(* Functionsblocks *************************************************)
	rTrigExecute											:	R_TRIG;
	SoERead													:	FB_SoERead_ByDriveRef	:= (tTimeOut := DEFAULT_ADS_TIMEOUT);
(*******************************************************************)
END_VAR
VAR CONSTANT
	ST_IDLE													:	INT := 0;
	ST_PEAKCURRENT											:	INT := 10;
	ST_COSPHI												:	INT := 20;
	ST_ERROR												:	INT := 998;
	ST_RESET												:	INT := 999;
	
	ERR_PEAKCURRENT											:	UDINT := 1;
	ERR_COSPHI												:	UDINT := 2;
END_VAR


(* Init drive ref **************************************************)
	IF AdsAddr.port <> SoERead.stDriveRef.nSlaveAddr
	THEN
		SoERead.stDriveRef.sNetId							:= F_CreateAmsNetId(AdsAddr.netId);
		SoERead.stDriveRef.nSlaveAddr						:= AdsAddr.port;
		SoERead.stDriveRef.nDriveNo							:= Channel;
	END_IF
(* calculate  ******************************************************)
	IF NOT busy
		AND MemParamSet = ActParameterSet
		AND Enable
	THEN
		AbsoluteCurrent										:= TO_REAL(_AbsoluteCurrent * (MemPeakCurrent / 1000)) / 1000;
		ApparentPower										:= SQRT(3) * TO_LREAL(AbsoluteCurrent * AbsoluteVoltage)  / 1000;
		ActivePower											:= ApparentPower * TO_LREAL(MemCosPhi) / 100.0;
		ReactivePower										:= SQRT(EXPT(ApparentPower,2) - EXPT(ActivePower,2));
	END_IF
(* Trigger Execute *************************************************)
	rTrigExecute(CLK := MemParamSet <> ActParameterSet AND Enable);
	
(* get params ******************************************************)
	CASE state OF
	ST_IDLE:	
		IF rTrigExecute.Q
		THEN
			State											:= ST_PEAKCURRENT;
		END_IF
	ST_PEAKCURRENT:	// read P-x-0092 configured peak current
		IF NOT SoERead.bBusy
			AND SoERead.bExecute
		THEN
			state											:= SEL(SoERead.bError, ST_COSPHI, 99);
			ErrorID											:= SEL(SoERead.bError, 0, ERR_PEAKCURRENT);
			ErrorText										:= SEL(SoERead.bError, '', 'Fehler beim Lesen vom Kanal Spitzenstrom');
		END_IF
		SoERead(
			stDriveRef	:= ,  //See init for drive ref
			nIdn		:= Get_P_WORD(ActParameterSet) + 092,
			nElement	:= EC_SOE_ELEMENT_VALUE (* 16#40*),
			pDstBuf		:= ADR(MemPeakCurrent),
			cbBufLen	:= SIZEOF(MemPeakCurrent),
			bExecute	:= State = 10,
			tTimeout	:= ,
			bBusy		=> ,
			bError		=> ,
			iAdsErrId	=> ,
			iSercosErrId=> ,
			dwAttribute	=> );
	ST_COSPHI:	// read P-x-0104 cos phi
		IF NOT SoERead.bBusy
			AND SoERead.bExecute
		THEN
			MemParamSet										:= SEL(SoERead.bError, ActParameterSet, MemParamSet);
			state											:= SEL(SoERead.bError, ST_IDLE, ST_ERROR);
			ErrorID											:= SEL(SoERead.bError, 0, ERR_COSPHI);
			ErrorText										:= SEL(SoERead.bError, '', 'Fehler beim Lesen vom cos phi Parameter');
		END_IF
		SoERead(
			stDriveRef	:= ,  //See init for drive ref
			nIdn		:= Get_P_WORD(ActParameterSet) + 104,
			nElement	:= EC_SOE_ELEMENT_VALUE (* 16#40*),
			pDstBuf		:= ADR(MemCosPhi),
			cbBufLen	:= SIZEOF(MemCosPhi),
			bExecute	:= State = 20,
			tTimeout	:= ,
			bBusy		=> ,
			bError		=> ,
			iAdsErrId	=> ,
			iSercosErrId=> ,
			dwAttribute	=> );
	ST_ERROR:			// wait till Error is quit
		IF ConfirmTrig
		THEN
			ErrorText										:= '';
			ErrorID											:= 0;
			state											:= ST_RESET;
		END_IF
	ST_RESET:		
		IF NOT SoERead.bBusy
			AND NOT SoERead.bError
		THEN
			state											:= ST_IDLE;
		END_IF
		SoERead(
			stDriveRef	:= ,  //See init for drive ref
			nIdn		:= Get_P_WORD(ActParameterSet) + 092,
			nElement	:= EC_SOE_ELEMENT_VALUE (* 16#40*),
			pDstBuf		:= ADR(MemPeakCurrent),
			cbBufLen	:= SIZEOF(MemPeakCurrent),
			bExecute	:= FALSE,
			tTimeout	:= ,
			bBusy		=> ,
			bError		=> ,
			iAdsErrId	=> ,
			iSercosErrId=> ,
			dwAttribute	=> );
	END_CASE
	
	Error		:= state = ST_ERROR;
	Busy		:= state <> 0 OR SoERead.bBusy;
(*******************************************************************)

METHOD PRIVATE get_P_WORD : WORD
VAR_INPUT
	SetNumber			:	INT;
END_VAR
(* Get P-Word dependent of parameter set *)
	IF SetNumber = 0 THEN
		Get_p_WORD			:= P_0_IDN;
	ELSIF SetNumber = 1 THEN
		Get_P_WORD			:= P_1_IDN;
	ELSIF SetNumber = 2 THEN
		Get_P_WORD			:= P_2_IDN;
	ELSIF SetNumber = 3 THEN
		Get_P_WORD			:= P_3_IDN;
	ELSIF SetNumber = 4 THEN
		Get_P_WORD			:= P_4_IDN;
	ELSIF SetNumber = 5 THEN
		Get_P_WORD			:= P_5_IDN;
	ELSIF SetNumber = 6 THEN
		Get_P_WORD			:= P_6_IDN;
	ELSIF SetNumber = 7 THEN
		Get_P_WORD			:= P_7_IDN;
	END_IF
END_METHOD

METHOD PRIVATE get_S_WORD : WORD
VAR_INPUT
	SetNumber			:	INT;
END_VAR
(* Get S-Word dependent of parameter set *)
	IF SetNumber = 0 THEN
		Get_S_WORD			:= S_0_IDN;
	ELSIF SetNumber = 1 THEN
		Get_S_WORD			:= S_1_IDN;
	ELSIF SetNumber = 2 THEN
		Get_S_WORD			:= S_2_IDN;
	ELSIF SetNumber = 3 THEN
		Get_S_WORD			:= S_3_IDN;
	ELSIF SetNumber = 4 THEN
		Get_S_WORD			:= S_4_IDN;
	ELSIF SetNumber = 5 THEN
		Get_S_WORD			:= S_5_IDN;
	ELSIF SetNumber = 6 THEN
		Get_S_WORD			:= S_6_IDN;
	ELSIF SetNumber = 7 THEN
		Get_S_WORD			:= S_7_IDN;
	END_IF
END_METHOD

END_FUNCTION_BLOCK

// POUs/IO/Drives/SoE/AxDriveSoE_Ax5000CommutationCalib
FUNCTION_BLOCK AxDriveSoE_Ax5000CommutationCalib EXTENDS FbBase
VAR CONSTANT
	STEP_COUNT											:	INT := 1;
	P150_NAMEPLATE_TYPE									:	E_AX5000_P_0150_DigitalNamePlate := E_AX5000_P_0150_DigitalNamePlate.EAX5000_P_0150_DIGITALNAMEPLATE_BECKHOFF; //1= Digital nameplate = Beckhoff
	P150_COMMUTATION_MODE_FEEDBACK						:	UINT := 1; //1= Feedback commutation offset
	
//	P150_NO_NAMEPLATE									:	UINT := 0; //0= Digital nameplate = no nameplate
//	P150_COMMUTATION_MODE_ADJUSTABLE					:	UINT := 3; //3= Adjustable mechanical offset 
END_VAR
VAR_OUTPUT CONSTANT
{attribute 'displaymode':='binary'}
	OPTION_READ_ONLY									:	BYTE  := 2#0000_0001; //Read actual commutation offset of the motor (not stored value in drive)
{attribute 'displaymode':='binary'}
	OPTION_P98_IS_EMPTY									:	BYTE  := 2#0000_0010; //Digital nameplate not initialized, skip check if entries. Select this option for first time setup
END_VAR
VAR_INPUT
	AdsAddr												: 	AMSADDR; //Terminal AMS Net Addr.	
	Channel												:	USINT;

{attribute 'displaymode':='binary'}         			
	Options												:	BYTE  := 2#0000_0000; (* Option constants are predefined, so they can accordingly be passed symbolically to the block 
																					.0 = TRUE read only 
																					*)

	
	MaxComPosDifference									:	LREAL := 15.0; //Maximal commutation position offset (Parameter P167, result of command P166)
END_VAR
VAR_IN_OUT
	axis												: AXIS_REF;
END_VAR
VAR_OUTPUT

	P0053												: AX5000_P_0053; // Configured motor type
	P0058												: AX5000_P_0058; // Mechanical commutation offset after command P166
	P0150												: AX5000_P_0150; // Feedback type form startup list
	P0167												: AX5000_P_0167; //Motor and feedback connection check parameter
	P0098												: AX5000_P_0098_beckhoff := (	
															Id_prat_1:= 1113940843,
															Id_prat_2:= 1752131174,	
														//	Name_plate_type := , 
															Version_no:=2,
															Motor_vendor:= 0, //None
															Serial_number:= 999999); //Digital nameplate
	Offset												:	LREAL; //Scaled value

	SercosErrId											: UDINT;
END_VAR
VAR
(*  Memory *****************************************************)
	lastState											: INT := 0;

(*  Timer ******************************************************)
(*  Trigger ****************************************************)

(*  Blocks *****************************************************)
	SoECommand 											: FB_SoEExecuteCommand 	:= (Timeout := t#30s);
	SoEWritePassword 									: FB_SoEWritePassword 	:= (Password :=(strData := 'AX5000', iActualSize := 128, iMaxSize := 128), Timeout := DEFAULT_ADS_TIMEOUT);
	SoEReset											: FB_SoEReset 			:= (Timeout := DEFAULT_ADS_TIMEOUT);
	SoEWrite											: FB_SoEWrite 			:= (Timeout := T#30S);
	SoERead												: FB_SoERead 			:= (Timeout := DEFAULT_ADS_TIMEOUT);
	
(*  Error ******************************************************)
(*  Dummys *****************************************************)
	{attribute 'hide' := ''}
	i,j													: INT := 0;

END_VAR

	(*********************************************************)
	
(* state machine ********************************************************)
	rtExecute(CLK := Execute);
	CASE state OF
	0 : 
		Busy 											:= FALSE;
		
		IF NOT Execute THEN
			Done 										:= FALSE;
			Error 										:= FALSE;
			ErrorID 									:= 0;
			SercosErrId									:= 0;
		END_IF
		IF rtExecute.Q THEN
			IF axis.status.ControlLoopClosed AND NOT Options.1 THEN
				Error 									:= TRUE;
				ErrorID 								:= 19266; //xis is enabled but should not be enabled for this process.

			ELSIF AdsAddr.netId[0] = 0
			THEN
 				Error 									:= TRUE;
				ErrorID 								:= 15; //Invalid AMS net id
	
			ELSIF AdsAddr.port = 0
			THEN
				Error 									:= TRUE;
				ErrorID 								:= 24; //Invalid ADS Port
						
			ELSE
				Busy									:= TRUE;	
				Done 									:= FALSE;
				Error 									:= FALSE;
				ErrorID 								:= 0;
				SercosErrId								:= 0;	
				
				Offset									:= 0.0;
				MEMSET(ADR(P0053),0,SIZEOF(P0053));
				MEMSET(ADR(P0058),0,SIZEOF(P0058));
				MEMSET(ADR(P0150),0,SIZEOF(P0150));
				MEMSET(ADR(P0167),0,SIZEOF(P0167));
				
				SoECommand(Execute := FALSE, Axis := axis);
				SoEWrite(Execute := FALSE, Axis := axis);
				SoERead(Execute := FALSE, Axis := axis);
				SoEReset(Execute := FALSE, Axis := axis);
				SoEWritePassword(Execute := FALSE, Axis := axis);
		
					
				state									:= state + STEP_COUNT;
			END_IF
		END_IF
	
	1:	(*write drive password *)
		SoEWritePassword(
			NetId:= , 
			Execute:=TRUE , 
			Timeout:= , 
			Password:= , //See declaration 
			Axis:=axis , 
			Busy=> , 
			Error=> , 
			AdsErrId=> , 
			SercosErrId=> );
	
		IF NOT SoEWritePassword.busy
		THEN
			IF SoEWritePassword.Error
			THEN
				Busy									:= FALSE;
				Error									:= TRUE;
				ErrorId									:= SoEWritePassword.AdsErrId;
				SercosErrId								:= SoEWritePassword.SercosErrId;
				state 									:= 0;
			ELSE
				
				state									:= state + STEP_COUNT;
			END_IF		
			SoEWritePassword(Execute := FALSE, Axis := axis);
		END_IF
			
	2:	(* Reset active errors *)
		SoEReset(
			NetId:= , 
			Execute:=TRUE , 
			Timeout:= , 
			Axis:=axis , 
			Busy=> , 
			Error=> , 
			AdsErrId=> , 
			SercosErrId=> );
			
		IF NOT SoEReset.Busy
		THEN
			IF SoEReset.Error
			THEN
				Busy									:= FALSE;
				Error									:= TRUE;
				ErrorId									:= SoEReset.AdsErrId;
				SercosErrId								:= SOEReset.SercosErrId;
				state 									:= 0;
			ELSE
				
				state									:= state + STEP_COUNT;
			END_IF	
			SoEReset(Execute := FALSE, Axis := axis);	
		END_IF

	3: // read configured motor type
		SoERead(
			NetId:= , 
			Idn:=P_0_IDN+53 , // IDN P-0-0053 Configured motor type
			Element:=EC_SOE_ELEMENT_VALUE , 
			pDstBuf:=ADR(P0053) , 
			BufLen:=SIZEOF(P0053) , 
			Execute:=TRUE , 
			Timeout:= , 
			Axis:=axis , 
			Busy=> , 
			Error=> , 
			AdsErrId=> , 
			SercosErrId=> , 
			Attribute=> );
			
		IF NOT SoERead.Busy
		THEN
			IF SoERead.Error
			THEN
				Busy									:= FALSE;
				Error									:= TRUE;
				ErrorId									:= SoERead.AdsErrId;
				SercosErrId								:= SoERead.SercosErrId;
				state 									:= 0;
			ELSE		
				
				state									:= state + STEP_COUNT;
			END_IF	
			SoERead(Execute := FALSE, Axis := axis);	
		END_IF
		
	4: //Read feedback type form startup list
		SoERead(
			NetId:= , 
			Idn:=P_0_IDN+150 , 
			Element:=EC_SOE_ELEMENT_VALUE , 
			pDstBuf:=ADR(P0150) , 
			BufLen:=SIZEOF(P0150) , 
			Execute:=TRUE , 
			Timeout:= , 
			Axis:=axis , 
			Busy=> , 
			Error=> , 
			AdsErrId=> , 
			SercosErrId=> , 
			Attribute=> );
			
		IF NOT SoERead.Busy
		THEN
			IF SoERead.Error
			THEN
				Busy									:= FALSE;
				Error									:= TRUE;
				ErrorId									:= SoERead.AdsErrId;
				SercosErrId								:= SoERead.SercosErrId;
				state 									:= 0;
			ELSE				
				state									:= state + STEP_COUNT;
			END_IF		
			SoERead(Execute := FALSE, Axis := axis);
		END_IF		
		
	5: (* Reserved *****************************************************)
		state											:= state + STEP_COUNT;
		
	6: //Read nameplate to check content (must be initialized) *************************
		SoERead(
			NetId:= , 
			Idn:=P_0_IDN+98 , 
			Element:=EC_SOE_ELEMENT_VALUE , 
			pDstBuf:=ADR(P0098) , 
			BufLen:=SIZEOF(P0098) , 
			Execute:=TRUE, 
			Timeout:= , 
			Axis:=axis , 
			Busy=> , 
			Error=> , 
			AdsErrId=> , 
			SercosErrId=> , 
			Attribute=> );	
		
		IF NOT SoERead.Busy
		THEN
			IF SoERead.Error
			THEN
				Busy									:= FALSE;
				Error									:= TRUE;
				ErrorId									:= SoERead.AdsErrId;
				SercosErrId								:= SoERead.SercosErrId;
				state 									:= 0;
			ELSE
				Offset									:= TO_LREAL(P0098.Position_offset) * 0.01;
				SoERead(Execute := FALSE, Axis := axis);	
				//Check parameter of P150
				IF Options.0
				THEN //Read only
					Busy								:= FALSE;
					Done								:= TRUE;
					state 								:= 0;
					
				ELSIF Options.1
				THEN //Nameplate not active, ignore current setting
					state								:= 10;	
					
				ELSIF TO_UINT(P0150.ParameterChannel.CommutationMode0) <> P150_COMMUTATION_MODE_FEEDBACK 
				THEN
					Busy								:= FALSE;
					Error								:= TRUE;
					ErrorId								:= E_AdsErr.DEVICE_INVALIDPARM;
					SercosErrId							:= 16#F749; //Feedback parameter invalid
					state 								:= 0;	
				ELSIF P0150.ParameterChannel.DigitalNamePlate <> P150_NAMEPLATE_TYPE
				THEN
					Busy								:= FALSE;
					Error								:= TRUE;
					ErrorId								:= E_AdsErr.DEVICE_INVALIDPARM;
					SercosErrId							:= 16#F749; //Invalid nameplate
					state 								:= 0;			
			
				ELSIF P0098.Name_plate_type <> P0150.ParameterChannel.DigitalNamePlate 
				THEN
					Busy								:= FALSE;
					Error								:= TRUE;
					ErrorId								:= E_AdsErr.DEVICE_INVALIDPARM;
					SercosErrId							:= 16#F803; //Unknow nameplate
					state 								:= 0;					
				
				ELSIF P0098.Position_offset = 0.0 
				THEN
					Busy								:= FALSE;
					Error								:= TRUE;
					ErrorId								:= E_AdsErr.DEVICE_INVALIDPARM;
					SercosErrId							:= 16#F742; //Invalid commutation offset
					state 								:= 0;
						
				ELSIF P0098.Feedback_typ <> P0150.FeedbackTypeString 
				THEN
					Busy								:= FALSE;
					Error								:= TRUE;
					ErrorId								:= E_AdsErr.DEVICE_INVALIDPARM;
					SercosErrId							:= 16#F708; //Feedback type invalid
					state 								:= 0;		
				ELSIF P0098.Motor_type <> P0053.Configures_motor_type 
				THEN
					Busy								:= FALSE;
					Error								:= TRUE;
					ErrorId								:= E_AdsErr.DEVICE_INVALIDPARM;
					SercosErrId							:= 16#FD09; //Motor type invalid
					state 								:= 0;				
				ELSE
					state								:= 10;	
				END_IF	
			END_IF
		END_IF
		
	10:	// Start command P-0-0160 - calibrate commutation offset ***********************************************	
		SoECommand(
			NetId:='' , 
			Idn:=P_0_IDN+160 , //command P-0-0160 = calibrate commutation offset 
			Execute:= TRUE, 
			Timeout:= , 
			Axis:=axis , 
			Busy=> , 
			Error=> , 
			AdsErrId=> , 
			SercosErrId=> );
		
		IF NOT SoECommand.Busy
		THEN
			IF SoECommand.Error
			THEN
				Busy									:= FALSE;
				Error									:= TRUE;
				ErrorId									:= SoECommand.AdsErrId;
				SercosErrId								:= SoECommand.SercosErrId;
				state 									:= 0;
			ELSE
				state									:= state + STEP_COUNT;
			END_IF		
			SoECommand(Execute := FALSE, Axis := axis);
		END_IF
	
	11: // read mechanical commutation offset result of command P160
		SoERead(
			NetId:= , 
			Idn:=P_0_IDN+58 , // IDN P-0-0167 = parameters to check commutation and rotation direction
			Element:=EC_SOE_ELEMENT_VALUE , 
			pDstBuf:=ADR(P0058) , 
			BufLen:=SIZEOF(P0058) , 
			Execute:= TRUE , 
			Timeout:= , 
			Axis:=axis , 
			Busy=> , 
			Error=> , 
			AdsErrId=> , 
			SercosErrId=> , 
			Attribute=> );	
		
		IF NOT SoERead.Busy
		THEN
			IF SoERead.Error
			THEN
				Busy									:= FALSE;
				Error									:= TRUE;
				ErrorId									:= SoERead.AdsErrId;
				SercosErrId								:= SoERead.SercosErrId;
				state 									:= 0;
			ELSE
				//Init nameplate information - see also declaration
				P0098.Motor_type						:= P0053.Configures_motor_type;
				P0098.Feedback_typ						:= P0150.FeedbackTypeString;	
				P0098.Name_plate_type					:= P0150.ParameterChannel.DigitalNamePlate;
				P0098.Position_offset					:= P0058.Mechanical_commutation_offset;
				Offset									:= TO_LREAL(P0058.Mechanical_commutation_offset) * 0.01;		
	
				state									:= state + STEP_COUNT;
			END_IF	
			SoERead(Execute := FALSE, Axis := axis);	
		END_IF
		
	12: // Start command P-0-0166 - Motor and feedback connection check 
		SoECommand(
			NetId:='' , 
			Idn:=P_0_IDN+166 , //command P-0-0166 = motor and feedback connection check 
			Execute:= TRUE, 
			Timeout:= , 
			Axis:=axis , 
			Busy=> , 
			Error=> , 
			AdsErrId=> , 
			SercosErrId=> );
		
		IF NOT SoECommand.Busy
		THEN
			IF SoECommand.Error
			THEN
				Busy									:= FALSE;
				Error									:= TRUE;
				ErrorId									:= SoECommand.AdsErrId;
				SercosErrId								:= SoECommand.SercosErrId;
				state 									:= 0;
			ELSE
				
				state									:= state + STEP_COUNT;
			END_IF		
			SoECommand(Execute := FALSE, Axis := axis);
		END_IF
	
	13: // read P-0-0167 read connection check results
		SoERead(
			NetId:= , 
			Idn:=P_0_IDN+167 , // IDN P-0-0167 = parameters to check commutation and rotation direction
			Element:=EC_SOE_ELEMENT_VALUE , 
			pDstBuf:=ADR(P0167) , 
			BufLen:=SIZEOF(P0167) , 
			Execute:= TRUE , 
			Timeout:= , 
			Axis:=axis , 
			Busy=> , 
			Error=> , 
			AdsErrId=> , 
			SercosErrId=> , 
			Attribute=> );
				
		IF NOT SoERead.Busy
		THEN
			IF SoERead.Error
			THEN
				Busy									:= FALSE;
				Error									:= TRUE;
				ErrorId									:= SoERead.AdsErrId;
				SercosErrId								:= SoERead.SercosErrId;
				state 									:= 0;
			ELSE				
				IF P0167.EqualDirektions <> 1
					OR
					TO_LREAL(P0167.Commutation_position_difference) * 0.01 > MaxComPosDifference 
					AND TO_LREAL(P0167.Commutation_position_difference) * 0.01 < 360.0 - MaxComPosDifference
				THEN
					Busy								:= FALSE;
					Error								:= TRUE;
					ErrorId								:= E_AdsErr.DEVICE_INVALIDPARM;
					SercosErrId							:= 16#F702; //Feedback position invalid
					state 								:= 0;
				ELSE                                	
					state								:= state + STEP_COUNT;
				END_IF
			END_IF		
			SoERead(Execute := FALSE, Axis := axis);
		END_IF
		
	14:	// Write digital motor plate with commutation offset
		SoEWrite(
			NetId:= , 
			Idn:=P_0_IDN+98, // P0-0-0098 = digital motor plate 
			Element:=EC_SOE_ELEMENT_VALUE , 
			pSrcBuf:=ADR(P0098) ,
			BufLen:=SIZEOF(P0098) ,
			Execute:=TRUE,
			Timeout:= , 
			Password:= SoEWritePassword.Password, 
			Axis:=axis , 
			Busy=> , 
			Error=> , 
			AdsErrId=> , 
			SercosErrId=> );
			
		IF NOT SoEWrite.Busy
		THEN
			IF SoEWrite.Error
			THEN
				Busy									:= FALSE;
				Error									:= TRUE;
				ErrorId									:= SoEWrite.AdsErrId;
				SercosErrId								:= SoEWrite.SercosErrId;
				state 									:= 0;
			ELSE
				
				state									:= state + STEP_COUNT;
			END_IF	
			SoEWrite(Execute := FALSE, Axis := axis);	
		END_IF

	15: // Command P-0-0162 - Save digital name plate
		SoECommand(
			NetId:= , 
			Idn:=P_0_IDN+162 , //save digital name plate 
			Execute:=TRUE , 
			Timeout:= , 
			Axis:=axis , 
			Busy=> , 
			Error=> , 
			AdsErrId=> , 
			SercosErrId=> );
	
		IF NOT SoECommand.Busy
		THEN
			IF SoECommand.Error
			THEN
				Busy									:= FALSE;
				Error									:= TRUE;
				ErrorId									:= SoECommand.AdsErrId;
				SercosErrId								:= SoECommand.SercosErrId;
				state 									:= 0;
			ELSE
				
				state									:= state + STEP_COUNT;
			END_IF		
			SoECommand(Execute := FALSE, Axis := axis);
		END_IF

	16: // Write digital motor plate with commutation offset again
		SoEWrite(
			NetId:= , 
			Idn:=P_0_IDN+98 , 
			Element:=EC_SOE_ELEMENT_VALUE , 
			pSrcBuf:=ADR(P0098) ,
			BufLen:=SIZEOF(P0098) ,
			Execute:= TRUE,
			Timeout:= , 
			Password:=SoEWritePassword.Password  , 
			Axis:=axis , 
			Busy=> , 
			Error=> , 
			AdsErrId=> , 
			SercosErrId=> );
				
		IF NOT SoEWrite.Busy
		THEN
			IF SoEWrite.Error
			THEN
				Busy									:= FALSE;
				Error									:= TRUE;
				ErrorId									:= SoEWrite.AdsErrId;
				SercosErrId								:= SoEWrite.SercosErrId;
				state 									:= 0;
			ELSE
				
				state									:= state + STEP_COUNT;
			END_IF	
			SoEWrite(Execute := FALSE, Axis := axis);	
		END_IF

	17: //Start command P-0-0161 - Save commutation offset in feedback 1
		SoECommand(
			NetId:= , 
			Idn:=P_0_IDN+161 , //save commutation offset 
			Execute:=TRUE , 
			Timeout:= , 
			Axis:=axis , 
			Busy=> , 
			Error=> , 
			AdsErrId=> , 
			SercosErrId=> );
		
		IF NOT SoECommand.Busy
		THEN
			IF SoEWrite.Error
			THEN
				Busy									:= FALSE;
				Error									:= TRUE;
				ErrorId									:= SoEWrite.AdsErrId;
				SercosErrId								:= SoEWrite.SercosErrId;
				state 									:= 0;
			ELSE
				Busy									:= FALSE;
				Done									:= TRUE;
				state 									:= 0;					
			END_IF		
			SoECommand(Execute := FALSE, Axis := axis);
		END_IF
	
	ELSE
		;
	END_CASE

(* Record last state ******************************************)
IF state <> lastState AND state <> 0 AND NOT Error
THEN 
	lastState											:= state;
END_IF

(*************************************************************)

{attribute 'monitoring' := 'call'}
PROPERTY PUBLIC optP98IsEmpty : BOOL
GET
optP98IsEmpty := Options.1;
END_GET
SET
Options.1 := optP98IsEmpty;
END_SET
END_PROPERTY

{attribute 'monitoring' := 'call'}
PROPERTY PUBLIC optReadOnly : BOOL
GET
optReadOnly := Options.0;
END_GET
SET
Options.0 := optReadOnly;
END_SET
END_PROPERTY

END_FUNCTION_BLOCK

// POUs/IO/Drives/SoE/AxDriveSoE_Ax5000Param
{attribute 'no_check'}
//FB template to read and write parameter
//The FB can be enherided and derivatived methods of SeqRead/SeqWrite used for application specific parameter.
//The extended methods need to call the super class at the beginning and return true if execution will be finished. The allowed states for new parameter are 1..99
FUNCTION_BLOCK AxDriveSoE_Ax5000Param EXTENDS AxRWParaBase
VAR_OUTPUT CONSTANT
END_VAR 
VAR_INPUT                               					
	AdsAddr													: 	AMSADDR; //Terminal AMS Net Addr. 
	Channel													:	USINT := 0; //Drive channel 0 or 1 for a two channel AX5000
	SetKvPosition											:	LREAL; //S-0-0104 (rad/s)rad - e.g. 10.0		
	SetKpVelocity											:	LREAL; //S-0-0100 mA/(rad/s) - e.g. 0.058	
	SetTnVelocity											:	LREAL; //S-0-0101 0.1ms 		- e.g. 0.015	
END_VAR 
VAR_IN_OUT
END_VAR                               					
VAR_OUTPUT 	
//	MotorSN													:	STRING(15); 
	KvPosition												:	LREAL;//S-0-0104
	KpVelocity												:	LREAL;//S-0-0100
	TnVelocity												:	LREAL;//S-0-0101
	NominalMainVoltage										:	LREAL;//P-0-0201 Volt 
	ConfiguredChnPeakForce									:	LREAL;//P-0-0094 Nm                    										
	ErrorSoEId												:	UDINT := 0;
END_VAR                         	
VAR
(* Cache ************************************************************)

	
(* Trigger **********************************************************)

(* Timer ******************************************************************)

(* FBs ***************************************************************)
	SoEWrite												: 	FB_SoEWrite_ByDriveRef := (tTimeout := DEFAULT_ADS_TIMEOUT); //SoE read
	SoERead													: 	FB_SoERead_ByDriveRef := (tTimeout := DEFAULT_ADS_TIMEOUT); //SoE wriet

(* Dummy memory **********************************************************)

END_VAR

	(* Read/Write drive parameter														*)
	(************************************************************************************)
	
(* Execute ***************************************************************************************)
	SUPER^();
	
(*************************************************************************************************)

PROPERTY PROTECTED deviceAddrIsValid : BOOL
GET
deviceAddrIsValid := AdsAddr.port > 0;
END_GET
END_PROPERTY

METHOD PROTECTED getValue : BOOL //Return value = TRUE if execution finished and state incremented 
VAR_INPUT
	Idn							:	WORD;
	Element						:	BYTE;
	Len							:	UDINT;
	pActValue					:	PVOID; //Address of variable for actual value
	pSetValue					:	PVOID; //Address of variable for ser value variable, can be zero if no corresponding SetVariable exists
END_VAR

SoERead(bExecute := TRUE, nIdn := Idn, nElement := Element, pDstBuf := pActValue, cbBufLen := Len);
IF NOT SoERead.bBUSY 	
THEN
	IF NOT SoERead.bError
	THEN
		IF pSetValue <> 0 THEN MEMCPY(pSetValue, pActValue, Len); END_IF
		state 												:= state + 1; 
	ELSE
		Busy												:= FALSE;
		Error												:= TRUE;
		ErrorId												:= SoERead.iAdsErrId;
		ErrorSoEId											:= SoERead.iSercosErrId;
		ErrorText											:= CONCAT('Error read parameter in state:' , TO_STRING(state * -1));
		ErrorText											:= CONCAT(ErrorText , CONCAT(' Id:',TO_STRING(ErrorId)));
		ErrorText											:= CONCAT(ErrorText , CONCAT(' Sercos Err :',TO_STRING(ErrorSoEId)));
		State												:= 9999;
	END_IF
	SoERead(bExecute := FALSE);
	getValue												:= TRUE;
END_IF
END_METHOD

METHOD PROTECTED seqRead : BOOL //Return value = TRUE if execution finished 
VAR_IN_OUT
	State							:	INT;
END_VAR

(* Sequence read parameter **********************************)
	CASE state OF
	1..99: //Read application specific parameter  
		SeqRead												:= TRUE;
		
	1001: (* Init step ******************************************************)		
		SoERead(bExecute:=FALSE);
		IF NOT SoERead.bBusy
		THEN
			SoERead.stDriveRef.sNetId						:= F_CreateAmsNetId(AdsAddr.netId);	
			SoERead.stDriveRef.nSlaveAddr 					:= AdsAddr.port;
			SoERead.stDriveRef.nDriveNo 					:= TO_BYTE(Channel);			
			state											:= state + 1;	
		END_IF
		
	1002: (* Kv Position *************************************************************************************)
		IF getValue(Idn:= S_0_IDN + 104,	Element := EC_SOE_ELEMENT_VALUE,	LEN := SIZEOF(_UINT),		pActValue := ADR(_UINT),	pSetValue := 0 )
		THEN
			KvPosition	:= SetKvPosition					:= SEL(Error, TO_LREAL(_UINT) * 0.01, 0.0); 
		END_IF

	1003: (* Kp velocity *******************************************)
		IF getValue(Idn:= S_0_IDN + 100,	Element := EC_SOE_ELEMENT_VALUE,	LEN := SIZEOF(_UDINT),		pActValue := ADR(_UDINT),	pSetValue := 0 )
		THEN
			KpVelocity := SetKpVelocity						:= SEL(Error, TO_LREAL(_UDINT) * 0.001, 0.0);
		END_IF

	1004: (* Tn velocity ********************************************)
		IF getValue(Idn:= S_0_IDN + 101,	Element := EC_SOE_ELEMENT_VALUE,	LEN := SIZEOF(_UINT),		pActValue := ADR(_UINT),	pSetValue := 0 )
		THEN
			TnVelocity	:= SetTnVelocity					:= SEL(Error, TO_LREAL(_UINT) * 0.1, 0.0);
		END_IF
					
	1005: (* Nominal main voltage  ********************************************)
  		IF getValue(Idn:= P_0_IDN + 201,	Element := EC_SOE_ELEMENT_VALUE,	LEN := SIZEOF(_UINT),		pActValue := ADR(_UINT),	pSetValue := 0 )
		THEN
			NominalMainVoltage								:= SEL(Error, TO_LREAL(_UINT) * 0.1, 0.0);
		END_IF	
		
	1006: (* Configured Channel Peak Current ********************************************)
  		IF getValue(Idn:= P_0_IDN + 94,		Element := EC_SOE_ELEMENT_VALUE,	LEN := SIZEOF(_UDINT),		pActValue := ADR(_UDINT),	pSetValue := 0 )
		THEN
			ConfiguredChnPeakForce 							:= SEL(Error, TO_LREAL(_UDINT) * 0.01, 0.0);
		END_IF
	ELSE
		state												:= 1;
	END_CASE

(***********************************************************************************)
END_METHOD

METHOD PROTECTED seqWrite : BOOL //Return value = TRUE if execution finished 
VAR_IN_OUT
	State							:	INT;
END_VAR
(* Sequence write parameter *********************************************)
	CASE state OF
	1..99: //Write application specific parameter  
		SeqWrite											:= TRUE;
		
	1001: (* Init step ******************************************************)		
		SoEWrite(bExecute:= TRUE);
		IF NOT SoEWrite.bBusy
		THEN
			SoEWrite.stDriveRef.sNetId						:= F_CreateAmsNetId(AdsAddr.netId);	
			SoEWrite.stDriveRef.nSlaveAddr 					:= AdsAddr.port;
			SoEWrite.stDriveRef.nDriveNo 					:= Channel;		
			state											:= state + 1;	
		END_IF
	
	1002: (* Kv position *************************************************************************************)
		_UINT												:= TO_UINT(SetKvPosition * 100.0);
		IF setValue(Idn := S_0_IDN + 104, Element := EC_SOE_ELEMENT_VALUE,	LEN := SIZEOF(_UINT),		pActValue := 0,		pSetValue := ADR(_UINT) )
		THEN
			KvPosition										:= SetKvPosition;
		END_IF		
		
	1003: (* Kp velocity ****************************************)
		_UDINT												:= TO_UDINT(SetKpVelocity * 1000.0);
		IF setValue(Idn := S_0_IDN + 100, Element := EC_SOE_ELEMENT_VALUE,	LEN := SIZEOF(_UDINT),		pActValue := 0,		pSetValue := ADR(_UDINT) )
		THEN
			KpVelocity										:= SetKpVelocity;
		END_IF	
		
	1004: (* Tn velocity **********************************)
		_UINT											:= TO_UINT(SetTnVelocity * 10.0);
		IF setValue(Idn := S_0_IDN + 101, Element := EC_SOE_ELEMENT_VALUE,	LEN := SIZEOF(_UINT),		pActValue := 0,		pSetValue := ADR(_UINT) )
		THEN
			TnVelocity										:= SetTnVelocity;
		END_IF		ELSE
		state												:= 1;
	END_CASE

(************************************************************************************)
END_METHOD

METHOD PROTECTED setValue : BOOL //Return value = TRUE if execution finished and state incremented 
VAR_INPUT
	Idn							:	WORD;
	Element						:	BYTE;
	Len							:	UDINT;
	pActValue					:	PVOID; //Address of variable for actual value, can be zero if no corresponding acual value variable exists
	pSetValue					:	PVOID; //Address of variable for set value variable
END_VAR

IF pActValue <> 0 AND pSetValue <> 0 AND_THEN MEMCMP(pSetValue, pActValue, Len) = 0
THEN //Skip write parameter if set and actual value are equel
	state													:= state + 1;	
	setValue												:= TRUE;
ELSE
	SoEWrite(bExecute:= TRUE, nIdn := Idn, nElement := Element, pSrcBuf := pSetValue, cbBufLen := LEN);
	IF NOT SoEWrite.bBusy
	THEN
		IF NOT SoEWrite.bError
		THEN
			IF pActValue <> 0 THEN MEMCPY(pActValue, pSetValue, Len); END_IF	
			state											:= state + 1;
		ELSE
			Busy											:= FALSE;
			Error											:= TRUE;
			ErrorId											:= SoEWrite.iAdsErrId;
			ErrorSoEId										:= SoEWrite.iSercosErrId;
			ErrorText										:= CONCAT('Error write parameter in state:' , TO_STRING(state * -1));
			ErrorText										:= CONCAT(ErrorText , CONCAT(' Id:',TO_STRING(ErrorId)));
			ErrorText										:= CONCAT(ErrorText , CONCAT(' Sercos Err :',TO_STRING(ErrorSoEId)));
			State											:= 9999;
		END_IF
		SoEWrite(bExecute := FALSE);
		setValue											:= TRUE;
	END_IF		
END_IF
END_METHOD

END_FUNCTION_BLOCK

// POUs/IO/Drives/SoE/AxDriveSoE_Ax5000SwitchParamSet
FUNCTION_BLOCK AxDriveSoE_Ax5000SwitchParamSet EXTENDS FbBase
VAR_INPUT
	rAxis													:	REFERENCE TO AXIS_REF := 0; 	// Axis Ref
	TimeOut													:	TIME := DEFAULT_ADS_TIMEOUT;	// Timeout time
	NewParamSet												:	INT;							// Value for new parameterset
END_VAR
VAR_IN_OUT	
(* important for function *)	
	AdsAddr													:	AMSADDR;						// AdsAddr of AX5000
	Channel													:	USINT;                          // Drive channel number
END_VAR
VAR_OUTPUT
	ErrorText												:	T_MaxString;					// Error Text
	ActParamSet												:	INT := -1; 						// Value of active parameter set
END_VAR
VAR
(* Memory **********************************************************)
	StartSwitchParamSet										:	INT := 0;
	
	CountError												:	USINT;
(* Timer ***********************************************************)
	TimerWait												:	TON;
	TimerTimeOut											:	TON;
	
(* Functionsblocks *************************************************)

	SoEWrite												:	FB_SoEWrite_ByDriveRef	:= (tTimeOut := DEFAULT_ADS_TIMEOUT);
	SoERead													:	FB_SoERead_ByDriveRef	:= (tTimeOut := DEFAULT_ADS_TIMEOUT);
(*******************************************************************)
END_VAR
VAR CONSTANT
	ST_IDLE													:	INT := 0;
	ST_REFRESH												:	INT := 10;
	ST_PRESELECT											:	INT := 100;
	ST_DISABLED												:	INT := 110;
	ST_RESETEXECUTE											:	INT := 120;
	ST_SETPARAM												:	INT := 130;
	ST_WAIT													:	INT := 140;
	ST_ERROR												:	INT := 998;
	ST_RESET												:	INT := 999;
	
	ERR_REFRESH												:	UDINT := 1;
	ERR_PRESELECT											:	UDINT := 2;
	ERR_TIMEOUT_DISABLED									:	UDINT := 3;
	ERR_RESETEXECUTE										:	UDINT := 4;
	ERR_EXECUTE												:	UDINT := 5;
	
	PT_WAIT_TIME											:	TIME := T#20MS;
END_VAR

(* abort function-call if the reference is invalid *****************)
	IF NOT __ISVALIDREF(rAxis) THEN
		Busy												:= NOT Error;
		Error												:= TRUE;
		ErrorId												:= 16#4B30;
		ErrorText											:= 'Referenz rAxis invalid (0)';
		RETURN;
	END_IF

(* Init drive ref **************************************************)
	IF AdsAddr.port <> SoERead.stDriveRef.nSlaveAddr
	THEN
		SoERead.stDriveRef.sNetId							:= F_CreateAmsNetId(AdsAddr.netId);
		SoERead.stDriveRef.nSlaveAddr						:= AdsAddr.port;
		SoERead.stDriveRef.nDriveNo							:= Channel;
		
		SoEWrite.stDriveRef									:= SoERead.stDriveRef;
	END_IF
(* Trigger Execute *************************************************)
	rtExecute(CLK := Execute);
	
(* switch parameter set ********************************************)
	CASE State OF
	ST_IDLE:			// wait for command
	(* Get actual parameter set after restart *)
		IF ActParamSet < 0 
		THEN
			State											:= ST_REFRESH;
	(* Start switch parameter set *)
		ELSIF rtExecute.Q
		THEN
			setNewParam(NewParamSet);
		ELSIF NOT Execute
		THEN
			Error											:= FALSE;
			Done											:= FALSE;
			Busy											:= TRUE;
			ErrorId											:= 0;
			ErrorTExt										:= '';
		END_IF
		
	ST_REFRESH: 		// Refresh ActParamSet Variable
		IF NOT SoERead.bBusy
			AND SoERead.bExecute
		THEN
			State											:= SEL(SoERead.bError, ST_IDLE, ST_ERROR);
			Done											:= State = ST_IDLE;
			Error											:= State = ST_ERROR;	
			ErrorID											:= SEL(SoERead.bError, 0, ERR_REFRESH);
			ErrorText										:= SEL(SoERead.bError, '', 'Fehler beim Aktualisieren des aktuellen Parametersatzes');
		END_IF
		
		SoERead(
			stDriveRef	:= ,  //See init for drive ref
			nIdn		:= S_0_IDN + 254,
			nElement	:= EC_SOE_ELEMENT_VALUE (* 16#40*),
			pDstBuf		:= ADR(ActParamSet),
			cbBufLen	:= SIZEOF(ActParamSet),
			bExecute	:= State = ST_REFRESH,
			tTimeout	:= ,
			bBusy		=> ,
			bError		=> ,
			iAdsErrId	=> ,
			iSercosErrId=> ,
			dwAttribute	=> );
			
		ST_PRESELECT:		// Set New param value in drive preselection
			IF NewParamSet = ActParamSet
			THEN
				State										:= ST_IDLE;
			ELSIF NOT SoEWrite.bBusy
				AND SoEWrite.bExecute
			THEN
				State										:= SEL(SoEWrite.bError, ST_DISABLED, ST_ERROR);
				ErrorID										:= SEL(SoERead.bError, 0, ERR_PRESELECT);
				ErrorText									:= SEL(SoERead.bError, '', 'Fehler beim Schreiben der Vorwahl');
			END_IF
			
			SoEWrite(
				stDriveRef	:= ,  //See init for drive ref
				nIdn		:= S_0_IDN + 217,
				nElement	:= EC_SOE_ELEMENT_VALUE (* 16#40*),
				pSrcBuf		:= ADR(NewParamSet),
				cbBufLen	:= SIZEOF(NewParamSet),
				bExecute	:= State = ST_PRESELECT,
				tTimeout	:= ,
				bBusy		=> ,
				bError		=> ,
				iAdsErrId	=> ,
				iSercosErrId=> );
				
		ST_DISABLED:		// check if axis is disabled
			TimerTimeOut(IN := NOT rAxis.Status.Disabled, PT := TimeOut);
			IF TimerTimeOut.Q THEN
				TimerTimeOut(IN := FALSE);
				State											:= ST_ERROR;
				ErrorID											:= SEL(SoERead.bError, 0, ERR_TIMEOUT_DISABLED);
				ErrorText										:= SEL(SoERead.bError, '', 'Achse ist nicht deaktiviert');
			ELSIF rAxis.Status.Disabled THEN
				TimerTimeOut(IN := FALSE);
				State											:= ST_RESETEXECUTE;
			END_IF
		
		ST_RESETEXECUTE:	// reset the execute command in drive	
			StartSwitchParamSet									:= 0;
			IF NOT SoEWrite.bBusy
				AND SoEWrite.bExecute
			THEN
				State											:= SEL(SoEWrite.bError, ST_SETPARAM, ST_ERROR);
				ErrorID											:= SEL(SoERead.bError, 0, ERR_RESETEXECUTE);
				ErrorText										:= SEL(SoERead.bError, '', 'Fehler beim Zurücksetzen des Ausführungskomamando');
			END_IF
			SoEWrite(
				stDriveRef	:= ,  //See init for drive ref
				nIdn		:= S_0_IDN + 216,
				nElement	:= EC_SOE_ELEMENT_VALUE (* 16#40*),
				pSrcBuf		:= ADR(StartSwitchParamSet),
				cbBufLen	:= SIZEOF(StartSwitchParamSet),
				bExecute	:= State = ST_RESETEXECUTE,
				tTimeout	:= ,
				bBusy		=> ,
				bError		=> ,
				iAdsErrId	=> ,
				iSercosErrId=> );		
				
		ST_SETPARAM:		// Execute switch parameter set
			StartSwitchParamSet								:= 3;
			IF NOT SoEWrite.bBusy
				AND SoEWrite.bExecute
			THEN
				State										:= SEL(SoEWrite.bError, ST_WAIT, ST_ERROR);
				ErrorID										:= SEL(SoERead.bError, 0, ERR_EXECUTE);
				ErrorText									:= SEL(SoERead.bError, '', 'Fehler beim Setzen des Ausführungskommandos');
			END_IF
			SoEWrite(
				stDriveRef	:= ,  //See init for drive ref
				nIdn		:= S_0_IDN + 216,
				nElement	:= EC_SOE_ELEMENT_VALUE (* 16#40*),
				pSrcBuf		:= ADR(StartSwitchParamSet),
				cbBufLen	:= SIZEOF(StartSwitchParamSet),
				bExecute	:= State = ST_SETPARAM,
				tTimeout	:= ,
				bBusy		=> ,
				bError		=> ,
				iAdsErrId	=> ,
				iSercosErrId=> );
				
		ST_WAIT:			// wait a short time while the drive works with the command
			TimerWait(IN := TRUE, pt := PT_WAIT_TIME);
			IF TimerWait.Q THEN
				TimerWait(IN := FALSE);
				State										:= ST_REFRESH;
			END_IF
			
		ST_ERROR:			// wait till Error is quit
			IF TRUE
			THEN
				State										:= ST_RESET;
			END_IF
			
		ST_RESET:			// Reset Error			
			State											:= ST_IDLE;
			SoEWrite(
				stDriveRef	:= ,  //See init for drive ref
				nIdn		:= S_0_IDN + 216,
				nElement	:= EC_SOE_ELEMENT_VALUE (* 16#40*),
				pSrcBuf		:= ADR(StartSwitchParamSet),
				cbBufLen	:= SIZEOF(StartSwitchParamSet),
				bExecute	:= FALSE,
				tTimeout	:= ,
				bBusy		=> ,
				bError		=> ,
				iAdsErrId	=> ,
				iSercosErrId=> );
			SoERead(
				stDriveRef	:= ,  //See init for drive ref
				nIdn		:= S_0_IDN + 254,
				nElement	:= EC_SOE_ELEMENT_VALUE (* 16#40*),
				pDstBuf		:= ADR(ActParamSet),
				cbBufLen	:= SIZEOF(ActParamSet),
				bExecute	:= FALSE,
				tTimeout	:= ,
				bBusy		=> ,
				bError		=> ,
				iAdsErrId	=> ,
				iSercosErrId=> ,
				dwAttribute	=> );
	END_CASE
	Busy													:= State <> ST_IDLE ;
(*******************************************************************)

METHOD setNewParam : BOOL	// Result = Busy
VAR_INPUT
	ParamNo					:	INT;
END_VAR

	IF ParamNo <> ActParamSet
		AND State = ST_IDLE
	THEN
		Error											:= FALSE;
		Done											:= FALSE;
		Busy											:= TRUE;
		ErrorId											:= 0;
		ErrorTExt										:= '';
		NewParamSet 									:= ParamNo;
		TimerWait(IN := FALSE);
		TimerTimeOut(IN := FALSE);
		State											:= ST_PRESELECT;
	END_IF
	
	SetNewParam											:= State <> ST_IDLE;
END_METHOD

END_FUNCTION_BLOCK

// POUs/IO/Drives/SoE/AxDriveSoE_Ax5000wEvents
{attribute 'no_check'}
//AX5000 SoE status and diagnosis FB with eventlogger 
FUNCTION_BLOCK AxDriveSoE_Ax5000wEvents EXTENDS AxDriveSoE_Ax5000
VAR_INPUT
	EnableEvent												:	BOOL := TRUE;
	ConfirmTrig												:	BOOL ;
	SourceId												:	UDINT := 102000; //SoE Drive default multisource Id + Ax id
	Name													:	STRING(30) := '';
	ErrorLimitPos											:	BOOL := FALSE;
	ErrorLimitNeg											:	BOOL := FALSE;
END_VAR                 									
VAR_IN_OUT              									
END_VAR                 									
VAR_OUTPUT              	                    										
	EventStatus												:	DWORD;
	NoOfActiveEvents										:	INT;
	Error													: 	BOOL; //ADS error SoE FBs
{attribute 'displaymode':='hex'}
	ErrorId													:	UDINT; //ADS error id of SoE FBs
	ErrorText												: 	STRING(40);
END_VAR
VAR_OUTPUT CONSTANT
END_VAR
VAR

(* Zwischenspeicher *********************************************************************)


(* Timer ********************************************************************************)

(* Trigger ******************************************************************************)

(* Bausteine ****************************************************************************)
	Event													:	EventHandlingGrp10;

(* Dummy Speicher **********************************************************)
	i														: INT := 0 ;


(****************************************************************************)
END_VAR

	(************************************************************************************)
	(*																					*)
	(*		B E C K H O F F   N E W   A U T O M A T I O N   T E C H N O L O G Y    		*)
	(*																					*)
	(*		Eiserstr.5	D-33415 Verl	Germany	phone:	+49-5246-0	www.Beckhoff.Com	*)
    (*																					*)
    (*		Bausteinbeschreibung	:	AX5000 Drive Ctrl								*)
	(*		TwinCAT-Version			:	3.x or higher 									*)
	(*		Version					:	V3.0 											*)
 	(*		Autor					:	Daniel Schlingmann								*)
	(*		Lib						:	TcMc2Drive.lib / TcDrive.Lib					*)
	(*																					*)
	(************************************************************************************)

(* Trigger reset if by active quit **********)
	IF ConfirmTrig
	THEN
		confirm();
	END_IF

(* Call super *****************************)
	SUPER^();
	
(* Call events ****************************************************)
	_callEvents();

(******************************************************************************)

METHOD PRIVATE _callEvents : BOOL
VAR_INPUT
END_VAR

(* Check if msg activ and init some parameter ***********************)
	IF Event.no[1].Text2 <> Name AND Name <> '' OR Event.no[1].Text2 = '' AND rAxis.NcToPlc.AxisId <> 0
	THEN
		Event.no[1].eClass 									:= TC2_SYSTEM.TCEVENTCLASS_HINT;

		(* Init Name *)
		FOR i := Event.MIN_EVENT TO Event.MAX_EVENT DO
			Event.no[i].Text2								:= SEL(LEN(name)>1,CONCAT('Axis id:',DWORD_TO_STRING(rAxis.NcToPlc.AxisId)),name);
		END_FOR
	END_IF

(* workl Event Ctrl *************************************************)
	Event(
		ConfirmTrig := ConfirmTrig,
		Disable		:= rAxis.NcToPlc.AxisId = 0 OR NOT EnableEvent,
		SourceId	:= SourceId + rAxis.NcToPlc.AxisId,
		Status		=> EventStatus,
		NoOfActiveEvents => NoOfActiveEvents);

(* Error Hdl FB ******************************************************************)
	IF rAxis.Status.OpMode.SimulationAxis OR Event.confirmTrig
	THEN
		;
	ELSIF SoEDriveReset.bError
	THEN
		Error												:=	TRUE;
		ErrorId												:= 0;
		SercosErrorId										:= SoEDriveReset.iSercosErrId;
		ErrorText											:= CONCAT('SoeDrvReset SercosErrId: ',DWORD_TO_HEXSTR(SoEDriveReset.iSercosErrId,4,FALSE));
		ErrorText											:=	CONCAT(CONCAT(ErrorText,', ADSErrId: '),UINT_TO_STRING(SoEDriveReset.iAdsErrId));
	ELSIF SoEAX5000SetMotorCtrlWord.bError
	THEN
		Error												:=	TRUE;
		ErrorId												:= 0;
		SercosErrorId										:= SoEAX5000SetMotorCtrlWord.iSercosErrId;
		ErrorText											:= CONCAT('SoESetMotorCtrlWord SercosErrId: ',DWORD_TO_HEXSTR(SoEAX5000SetMotorCtrlWord.iSercosErrId,4,FALSE));
		ErrorText											:=	CONCAT(CONCAT(ErrorText,', ADSErrId: '),UINT_TO_STRING(SoEAX5000SetMotorCtrlWord.iAdsErrId));
	ELSIF SoERead.bError
	THEN
		Error												:=	TRUE;
		ErrorId												:= 0;
		SercosErrorId										:= SoERead.iSercosErrId;
		ErrorText											:= CONCAT('SoERead SercosErrId: ',DWORD_TO_HEXSTR(SoERead.iSercosErrId ,4,FALSE));
		ErrorText											:=	CONCAT(CONCAT(ErrorText,', ADSErrId: '),UINT_TO_STRING(SoERead.iAdsErrId));
	END_IF

(* Event Logger Meldungen *****************************************************)
	Event.no[1].Flag 										:= Status.bNotReadyToPowerUp;
	Event.no[2].Flag 										:= Status.bDrvShutdownBitC1D AND stateReadStatus = 0; Event.no[2].pText3 := ADR(DiagMsg.strData);
	Event.no[3].Flag 										:= FALSE;
	Event.no[4].Flag 										:= ErrorLimitPos;
	Event.no[5].Flag 										:= ErrorLimitNeg;
	Event.no[6].Flag 										:= SafetyError AND DiagNumber <> 16#0000_FDD9;
	Event.no[7].Flag 										:= FALSE;
	Event.no[8].Flag 										:= FALSE;
	Event.no[9].Flag 										:= FALSE;
	Event.no[10].Flag 										:= Error; Event.no[10].Text1 := TO_STRING(ErrorId);
	
(************************************************************************)
END_METHOD

METHOD PUBLIC confirm : BOOL //Return value = TRUE if busy
VAR_INPUT
END_VAR
Event.confirm();
Error												:= FALSE;
ErrorId												:= 0;
SercosErrorId										:= 0;
ErrorText											:= '';
		
confirm 											:= SUPER^.reset();
END_METHOD

END_FUNCTION_BLOCK

// POUs/IO/Drives/SoE/AxDriveSoE_Rexroth
{attribute 'no_check'}
//Bosch Rexroth EtherCAT SoE Drive Control
//based on Tc2_Drive
FUNCTION_BLOCK AxDriveSoE_Rexroth EXTENDS AxDriveBase
VAR_INPUT
	EnableEvent												:	BOOL := TRUE;
	ResetTrig												:	BOOL := FALSE; (* Quit event and reset drive (SoE Reset) *)
	SourceId												:	UDINT := 102000; //SoE Drive default multisource Id + Ax id
	Name													:	STRING(30) := '';
	ErrorLimitPos											:	BOOL := FALSE;
	ErrorLimitNeg											:	BOOL := FALSE;
	BreakUnlock												:	BOOL := FALSE; //Not implemented yet
	BreakLock												:	BOOL := FALSE; //Not implemented yet					
	SetReferenz												: 	BOOL := FALSE;
	Referenzpos												: 	LREAL := 0.0;
END_VAR                                 					
VAR_IN_OUT                              					
END_VAR                                 					
VAR_OUTPUT                                                					
	InReferenz												:	BOOL; (* Drive in reference *)
	RT_StatusChanged										:	BOOL;                                    						
	Status													:	ST_IndraDriveCsDriveStatus;
	C1D														:	ST_IndraDriveCs_C1D;
	DiagMsg 												: 	ST_SoE_String;
	DiagNumber 												: 	UDINT;
	Operational												: INPUT := (Force := TRUE);	(* Link to ALWAYS_TRUE or operational signal from drive *)
	EcState											AT %I* 	: 	UINT; (* Ethercat InfoData State *)
	SercosErrorId											:	UINT;                    					
	SafetyError										AT %I*	:	BOOL;	(* Ax5805 Drive Safety Error - Bit .7 in Input Safe Data Byte 0 oder 2 *)	
	EventStatus												:	DWORD;
	NoOfActiveEvents										:	INT;
	Busy													:	BOOL;
	Error													:	BOOL;
{attribute 'displaymode':='hex'}
	ErrorId													:	UDINT;
	ErrorText												:	STRING(40);
END_VAR                  						
VAR_OUTPUT CONSTANT
END_VAR
VAR (* EA Internal *)
	EcInfoDataState									AT %I* 	: 	UINT; (* Ethercat InfoData State *)
END_VAR
VAR

(* Cache *********************************************************************)
	MemDriveStatusword										: 	WORD;
	MEM_StatusTrig											:	BYTE;
	StatusTrig												:	BYTE;
	stateReadStatus											:	INT;
	stateCtrl												:	INT := 0;

(* Timer ********************************************************************************)

(* Trigger ******************************************************************************)

(* Instance ****************************************************************************)
	SoEDriveReset											: 	FB_SoEReset := (Timeout		:= DEFAULT_ADS_TIMEOUT);
	SoEWrite												: 	FB_SoEWrite := (Timeout		:= DEFAULT_ADS_TIMEOUT);
	SoERead													: 	FB_SoERead := (Timeout		:= DEFAULT_ADS_TIMEOUT);
	SoEExecuteCmd											:	FB_SoEExecuteCommand := (Timeout		:= DEFAULT_ADS_TIMEOUT);
	EcSetSlaveSTATE											:	FB_EcSetSlaveSTATE := (tTimeout		:= DEFAULT_ADS_TIMEOUT);
	Event													:	EventHandlingGrp10;

(* Dummy Speicher **********************************************************)
	i														: 	INT := 0 ;
	_word													:	WORD;
	_DWORD													:	DWORD;

(****************************************************************************)
END_VAR

	(************************************************************************************)
	(*																					*)
	(*		B E C K H O F F   N E W   A U T O M A T I O N   T E C H N O L O G Y    		*)
	(*																					*)
	(*		Eiserstr.5	D-33415 Verl	Germany	phone:	+49-5246-0	www.Beckhoff.Com	*)
    (*																					*)
    (*		Bausteinbeschreibung	:	Ethercat SoE MC2 Drive Ctrl						*)
	(*		TwinCAT-Version			:	3.x or higher	 								*)
	(*		Version					:	V3.0/05/11										*)
 	(*		Autor					:	Daniel Schlingmann								*)
	(*		Lib						:	TcMC2Drive.lib / TcDrive.Lib					*)
	(*																					*)
	(* Call cyclic																		*)
	(************************************************************************************)

(* abort function-call if the reference is invalid *****************************)
IF NOT __ISVALIDREF(rAxis)  
THEN
	Busy													:= NOT Error;
	Fault													:= TRUE;
	Ready													:= FALSE;
	Error													:= TRUE;
	ErrorId													:= 16#4B30;
	ErrorText												:= 'Referenz rAxis invalid (0)';
	SercosErrorId											:= 0;
	RETURN;
END_IF

(* DriveStatusword *****************************)
	Status 													:= F_ConvWordToSTIndraDriveCsDriveStatus(StatusWord);
	IF rAxis.Status.OpMode.SimulationAxis or AdsAddr.port = 0
	THEN
		Status.bNotReadyToPowerUp							:= FALSE;	
		Status.bDrvShutdownBitC1D							:= FALSE;
		Status.bReadyForEnable								:= TRUE;
		Status.bEnabled										:= TRUE;	
	END_IF
	
(* Drive Operation Input ***********************)
	Operational(
		Force		:= rAxis.Status.OpMode.SimulationAxis ,
		Invert		:= ,
		PT_ON		:= ,
		PT_OFF		:= ,
		Q_DIRECT	=> ,
		Q			=> ,
		Q_RT		=> ,
		Q_FT		=> );

(* DriveStatusBits ***********************************************)
	Fault													:= Status.bDrvShutdownBitC1D
																OR rAxis.NcToPlc.StateDWord.28 (* DriveDeviceError *)
																OR rAxis.NcToPlc.StateDWord.30; (* IODataInvalid *)
                                						
	Ready 													:= NOT Fault
																	AND(Status.bReadyForEnable OR Status.bEnabled)
																	AND Operational.Q;
  
	SwitchedOn												:= Status.bEnabled AND NOT Fault;	
	                              	
(* Reset Drive ****************************************************)
	SoEDriveReset(
		NetId		:= ,
		Execute		:= ,
		Timeout		:= ,
		Axis		:= rAxis,
		Busy		=> ,
		Error		=> ,
		AdsErrId	=> ,
		SercosErrId	=> );

	IF SoEDriveReset.Busy 
	THEN
		; (* Block ist currend working *)
	ELSIF ResetTrig
	THEN
		reset();
	ELSIF SoEDriveReset.Execute
	THEN
	(*	RefreshStatus();  *)
		SoEDriveReset.Execute 								:= FALSE;
	END_IF

(* Set Etehrcat State to OP ********************************************)
	EcSetSlaveSTATE(
		sNetId		:= F_CreateAmsNetId(nIds := AdsAddr.netId),
		nSlaveAddr	:= AdsAddr.port,
		bExecute	:= ,
		tTimeout	:= ,
		reqState	:= Tc2_EtherCAT.EC_DEVICE_STATE_OP,
		bBusy		=> ,
		bError		=> ,
		nErrId		=> ,
		currState	=> );

	IF EcSetSlaveSTATE.bBusy
	THEN
		; (* Block ist currend working *)
	ELSIF EcSetSlaveSTATE.bExecute
		AND NOT ResetTrig
	THEN
		RefreshStatus();
		EcSetSlaveSTATE.bExecute 							:= FALSE;
	END_IF

(* Referenzieren *******************************************************)
	CASE stateCtrl OF
	-1,0:
		IF SetReferenz AND NOT rAxis.Status.OpMode.SimulationAxis AND AdsAddr.port > 0
		THEN
			writeReferenz();
		ELSE
			stateCtrl										:= 0;
		END_IF

	1: (* Referezwert schreiben **************************************)
		IF NOT SoEWrite.Busy
			AND SoEWrite.Execute
		THEN
			IF SoEWrite.Error
			THEN
				stateCtrl 									:= 0;
			ELSE                							
				stateCtrl									:= 2;
			END_IF
		END_IF

		_DWORD 												:= LREAL_TO_UDINT(Referenzpos);

		SoEWrite(
			NetId		:= ,
			Idn			:= S_0_IDN + 52,
			Element		:= EC_SOE_ELEMENT_VALUE ,
			pSrcBuf		:= ADR(_DWORD),
			BufLen		:= SIZEOF(_DWORD),
			Execute		:= stateCtrl = 1,
			Timeout		:= ,
			Password	:= ,
			Axis		:= rAxis,
			Busy		=> ,
			Error		=> ,
			AdsErrId	=> ,
			SercosErrId	=> );

	2: (* commad for setting setvalue *)
		IF NOT SoEExecuteCmd.Busy
			AND SoEExecuteCmd.Execute
		THEN
			IF SoEExecuteCmd.Error
			THEN
				stateCtrl 									:= 0;
			ELSE
				RefreshStatus();
				IF NOT SetReferenz
				THEN
					stateCtrl 								:= 0;
				ELSE            							
					stateCtrl 								:= -1;
				END_IF
			END_IF
		END_IF

		SoEExecuteCmd(
			NetId		:= '',
			Idn			:= P_0_IDN + 12,
			Execute		:= stateCtrl = 2,
			Timeout		:= ,
			Axis		:= rAxis,
			Busy		=> ,
			Error		=> ,
			AdsErrId	=> ,
			SercosErrId	=> );
	ELSE
		;
	END_CASE


(* evaluate sercos DriveStatusword *********************************************************)
	RT_StatusChanged 										:= SHR(StatusWord,2) <> MemDriveStatusword;
	MemDriveStatusword 										:= SHR(StatusWord,2);

(* Start Read Drive status *****************************************************************)
	CASE stateReadStatus OF
	0:
		StatusTrig.0 										:= rAxis.NcToPlc.StateDWord.28; (* DriveDeviceError *)
		StatusTrig.1 										:= rAxis.NcToPlc.StateDWord.30; (* IODataInvalid *)
                                							
		IF NOT rAxis.Status.OpMode.SimulationAxis AND AdsAddr.port > 0
			AND(RT_StatusChanged OR MEM_StatusTrig <> StatusTrig)
		THEN
			RefreshStatus();
		ELSE
			;
		END_IF

	(* Read Class 1 Diag *********************************************************)
	10:
		IF NOT SoERead.Busy
			AND SoERead.Execute
		THEN
			IF SoERead.Error
			THEN
				stateReadStatus 							:= 0;
			ELSE                    						
				C1D 										:= F_ConvWordToSTIndraDriveCsC1D(_word);
				stateReadStatus 							:= stateReadStatus + 1;
			END_IF
		END_IF

		SoERead(
			NetId		:= ,
			Idn			:= S_0_IDN + 11,
			Element		:= EC_SOE_ELEMENT_VALUE,
			pDstBuf		:= ADR(_word),
			BufLen		:= SIZEOF(_word),
			Execute		:= stateReadStatus = 10,
			Timeout		:= ,
			Axis		:= rAxis,
			Busy		=> ,
			Error		=> ,
			AdsErrId	=> ,
			SercosErrId	=> ,
			Attribute	=> );

	(* S-0-0403 In Referenz ********************************************************)
	11:
		IF NOT SoERead.Busy
			AND SoERead.Execute
		THEN
			IF SoERead.Error
			THEN
				stateReadStatus 							:= 0;
			ELSE
				InReferenz 									:= _WORD.0 AND _WORD.1;
				stateReadStatus 							:= stateReadStatus + 1;
			END_IF
		END_IF

		SoERead(
			NetId		:= ,
			Idn			:= S_0_IDN + 403,
			Element		:= EC_SOE_ELEMENT_VALUE,
			pDstBuf		:= ADR(_word),
			BufLen		:= SIZEOF(_word),
			Execute		:= stateReadStatus = 11,
			Timeout		:= ,
			Axis		:= rAxis,
			Busy		=> ,
			Error		=> ,
			AdsErrId	=> ,
			SercosErrId	=> ,
			Attribute	=> );

			
	(* Diag Message *********************************************************)
	12:
		IF NOT SoERead.Busy
			AND SoERead.Execute
		THEN
			IF SoERead.Error
			THEN
				stateReadStatus 							:= 0;
			ELSE
				stateReadStatus 							:= stateReadStatus + 1;
			END_IF
		END_IF

		SoERead(
			NetId		:= ,
			Idn			:= S_0_IDN + 95,
			Element		:= EC_SOE_ELEMENT_VALUE (* 16#40*),
			pDstBuf		:= ADR(DiagMsg),
			BufLen		:= SIZEOF(DiagMsg),
			Execute		:= stateReadStatus = 12,
			Timeout		:= ,
			Axis		:= rAxis,
			Busy		=> ,
			Error		=> ,
			AdsErrId	=> ,
			SercosErrId	=> ,
			Attribute	=> );

	(* Diag Number *********************************************************)
	13:
		IF NOT SoERead.Busy
			AND SoERead.Execute
		THEN
			IF SoERead.Error
			THEN
				stateReadStatus 							:= 0;
			ELSE
				stateReadStatus 							:= stateReadStatus + 1;
			END_IF
		END_IF

		SoERead(
			NetId		:= ,
			Idn			:= S_0_IDN + 390,
			Element		:= EC_SOE_ELEMENT_VALUE (* 16#40*),
			pDstBuf		:= ADR(DiagNumber),
			BufLen		:= SIZEOF(DiagNumber),
			Execute		:= stateReadStatus = 13,
			Timeout		:= ,
			Axis		:= rAxis,
			Busy		=> ,
			Error		=> ,
			AdsErrId	=> ,
			SercosErrId	=> ,
			Attribute	=> );
			
	(* reading status finished ************************************************************)
	ELSE (* Case else *)
		stateReadStatus 									:= 0;
	END_CASE

(* Event Logger Meldungen *****************************************************)
	Event.no[1].Flag 										:= Status.bNotReadyToPowerUp;
	Event.no[2].Flag 										:= Status.bDrvShutdownBitC1D AND stateReadStatus = 0; Event.no[2].pText3 := ADR(DiagMsg.strData);
	Event.no[3].Flag 										:= FALSE;
	Event.no[4].Flag 										:= ErrorLimitPos;
	Event.no[5].Flag 										:= ErrorLimitNeg;
	Event.no[6].Flag 										:= FALSE; //SafetyError AND DiagNumber <> 16#0000_FDD9;
	Event.no[7].Flag 										:= FALSE;
	Event.no[8].Flag 										:= FALSE;
	Event.no[9].Flag 										:= FALSE;
	Event.no[10].Flag 										:= Error;

	(* Check if msg activ and init some parameter ***********************)
	IF Event.no[1].Text2 <> Name AND Name <> '' OR Event.no[1].Text2 = '' AND rAxis.NcToPlc.AxisId <> 0
	THEN
		Event.no[1].eClass 									:= TC2_SYSTEM.TCEVENTCLASS_HINT;

		(* Init Name *)
		FOR i := Event.MIN_EVENT TO Event.MAX_EVENT DO
			Event.no[i].Text2								:= SEL(LEN(name)>1,CONCAT('Axis id:',DWORD_TO_STRING(rAxis.NcToPlc.AxisId)),name);
		END_FOR
	END_IF

(* workl Event Ctrl *************************************************)
	Event(
		ConfirmTrig := ResetTrig,
		Disable		:= rAxis.NcToPlc.AxisId = 0 OR NOT EnableEvent,
		SourceId	:= SourceId + rAxis.NcToPlc.AxisId,
		Status		=> EventStatus,
		NoOfActiveEvents => NoOfActiveEvents);
				
(* Error Hdl FB ******************************************************************)
	IF SoEDriveReset.Error
	THEN
		Error												:=	TRUE;
		ErrorId												:= 0;
		SercosErrorId										:= SoEDriveReset.SercosErrId;
		ErrorText											:= CONCAT('SoeDrvReset SercosErrId: ',DWORD_TO_HEXSTR(SoEDriveReset.SercosErrId,4,FALSE));
		ErrorText											:=	CONCAT(CONCAT(ErrorText,', ADSErrId: '),UINT_TO_STRING(SoEDriveReset.AdsErrId));
	ELSIF SoEExecuteCmd.Error
	THEN
		Error												:=	TRUE;
		ErrorId												:= 0;
		SercosErrorId										:= SoEExecuteCmd.SercosErrId;
		ErrorText											:= CONCAT('SoEExecuteCmd SercosErrId: ',DWORD_TO_HEXSTR(SoEExecuteCmd.SercosErrId,4,FALSE));
		ErrorText											:=	CONCAT(CONCAT(ErrorText,', ADSErrId: '),UINT_TO_STRING(SoEExecuteCmd.AdsErrId));
	ELSIF SoERead.Error
	THEN
		Error												:=	TRUE;
		ErrorId												:= 0;
		SercosErrorId										:= SoERead.SercosErrId;
		ErrorText											:= CONCAT('SoERead SercosErrId: ',DWORD_TO_HEXSTR(SoERead.SercosErrId,4,FALSE));
		ErrorText											:=	CONCAT(CONCAT(ErrorText,', ADSErrId: '),UINT_TO_STRING(SoERead.AdsErrId));
	ELSIF SoEWrite.Error
	THEN
		Error												:=	TRUE;
		ErrorId												:= 0;
		SercosErrorId										:= SoEWrite.SercosErrId;
		ErrorText											:= CONCAT('SoEWrite SercosErrId: ',DWORD_TO_HEXSTR(SoEWrite.SercosErrId,4,FALSE));
		ErrorText											:=	CONCAT(CONCAT(ErrorText,', ADSErrId: '),UINT_TO_STRING(SoEWrite.AdsErrId));
	END_IF

(* FB is Busy *******************************************************************)
	Busy 													:= stateCtrl > 0
																OR SoEDriveReset.Busy
																OR stateReadStatus > 0;

(******************************************************************************)

METHOD PUBLIC refreshStatus : BOOL //Return value = TRUE if busy
VAR_INPUT
END_VAR
IF NOT __ISVALIDREF(rAxis)  
THEN
	Busy													:= NOT Error;
	Error													:= TRUE;
	ErrorId													:= 16#4B30;
	ErrorText												:= 'Referenz rAxis invalid (0)';
	SercosErrorId											:= 0;
ELSIF stateReadStatus = 0 
THEN
	Busy													:= TRUE;
	Error													:= FALSE;
	ErrorTExt												:= '';
	ErrorId													:= 0;
	SercosErrorId											:= 0;
	stateReadStatus 										:= 10;
	StatusTrig.0 											:= rAxis.NcToPlc.StateDWord.28; (* DriveDeviceError *)
	StatusTrig.1 											:= rAxis.NcToPlc.StateDWord.30; (* IODataInvalid *)
	MEM_StatusTrig 											:= StatusTrig;
	MEMSET(ADR(DiagMsg),0,SIZEOF(DiagMsg));
	SoERead(
		Execute := FALSE,
		Axis 	:= rAxis);
ELSE
	Busy													:= TRUE;
END_IF                              						
                                    						
RefreshStatus												:= Busy AND stateReadStatus > 0;
END_METHOD

METHOD PUBLIC reset : BOOL //Return value = TRUE if busy
VAR_INPUT
END_VAR
IF NOT SoEDriveReset.Execute
THEN
	Error													:=	FALSE;
	ErrorId													:= 0;
	SercosErrorId											:= 0;
	Errortext												:= '';
END_IF
EcSetSlaveSTATE.bExecute									:= NOT (( UINT_TO_WORD(EcState) AND Tc2_EtherCAT.EC_DEVICE_STATE_MASK ) = Tc2_EtherCAT.EC_DEVICE_STATE_OP)
																AND EcState > 0 AND NOT rAxis.Status.OpMode.SimulationAxis;
										
Busy														:= SoEDriveReset.Busy OR NOT SoEDriveReset.Execute;               							
SoEDriveReset.Execute										:= NOT SoEDriveReset.Busy AND NOT rAxis.Status.OpMode.SimulationAxis AND AdsAddr.port > 0;
reset													:= Busy;
END_METHOD

METHOD PUBLIC writeReferenz : BOOL //Return value = TRUE if busy
VAR_INPUT
END_VAR
IF NOT __ISVALIDREF(rAxis)  
THEN
	Busy													:= NOT Error;
	Error													:= TRUE;
	ErrorId													:= E_AdsErr.DEVICE_INVALIDPARM;
	ErrorText												:= 'Referenz rAxis invalid (0)';
	SercosErrorId											:= 0;
ELSIF stateCtrl = 0 
THEN
	ErrorText												:= '';
	Error													:=	FALSE;
	ErrorId													:= 0;
	SercosErrorId											:= 0;
	Busy													:= TRUE;
	stateCtrl 												:= 1;
	SoEWrite(Execute := FALSE, Axis := rAxis);
	SoEExecuteCmd(Execute := FALSE, Axis := rAxis);

END_IF                              						
                                    	
writeReferenz													:= Busy AND stateCtrl > 0;
END_METHOD

END_FUNCTION_BLOCK

// POUs/IO/Drives/Stepper/AxDriveStepper_wEvents
{attribute 'no_check'}
//Beckhoff Stepper terminal diag and diagnosis with eventlogger - extended from AxDriveStepper
//EventHandling instance use inside
FUNCTION_BLOCK AxDriveStepper_wEvents EXTENDS AxDriveStepper
VAR CONSTANT         	
END_VAR  
VAR_INPUT
	EnableEvent												:	BOOL := TRUE; //Enable to show events
	ConfirmTrig												:	BOOL := FALSE; //Quit events
	SourceId												:	UDINT := 102600; //MDP742 Stepper CoE Drive default multisource Id + Ax id
	Name													:	STRING(30) := '';
	ErrorLimitPos											:	BOOL := FALSE;
	ErrorLimitNeg											:	BOOL := FALSE;
END_VAR                     					
VAR_IN_OUT                  					
END_VAR                     					
VAR_OUTPUT                  					
 	EventStatus												:	DWORD;       
	NoOfActiveEvents										:	INT;                    					
END_VAR                     					                   					
VAR                         					
END_VAR
VAR

(* Cache *********************************************************************)
	
(* Timer ********************************************************************************)

(* Trigger ******************************************************************************)

(* Instance ****************************************************************************)
	Event													:	EventHandlingGrp10;
	
(* Dummy Speicher **********************************************************)
	i														: INT := 0 ;
END_VAR

	(* Stepper Drive Control with events												*)
	(************************************************************************************)

(* Call super **********************************************)
	SUPER^();
	
(* work events *******************************************)
	_callEvents();

(*******************************************************)

METHOD PRIVATE _callEvents : BOOL
VAR_INPUT
END_VAR

(* Check if msg activ and init some parameter ***********************)
	IF Event.no[1].Text2 <> Name AND Name <> '' OR Event.no[1].Text2 = '' AND rAxis.NcToPlc.AxisId <> 0
	THEN
		Event.no[1].eClass 									:= TC2_SYSTEM.TCEVENTCLASS_STATEINFO;
		Event.no[3].eClass 									:= TC2_SYSTEM.TCEVENTCLASS_MESSAGE;
		
		(* Init Achsname *)
		FOR i := Event.MIN_EVENT TO Event.MAX_EVENT DO
		(*	Event.no[i].Text1								:= '';*)
			Event.no[i].Text2								:= SEL(LEN(name)>1,CONCAT('Axis id:',DWORD_TO_STRING(rAxis.NcToPlc.AxisId)),name);
		END_FOR
	END_IF

(* workl Event Ctrl *************************************************)
	Event(
		ConfirmTrig := ConfirmTrig,
		Disable		:= rAxis.NcToPlc.AxisId = 0 OR NOT EnableEvent,
		SourceId	:= SourceId + rAxis.NcToPlc.AxisId,
		Status		=> EventStatus,
		NoOfActiveEvents => NoOfActiveEvents);

(* Event Logger Meldungen *****************************************************)
	Event.no[1].Flag 										:= NOT Status_ReadyToEnable ; 
	Event.no[2].Flag 										:= Fault;
	Event.no[3].Flag 										:= (Status_Warning OR Diag_Configuration) AND NOT rAxis.Status.Homing AND rAxis.Status.Operational; //Avoid warning if drive is disabled (EL7037 and older FW on EL7047 <=06 - 2020-03-26) 				
	Event.no[4].Flag 										:= Diag_TorqueOverloaded;
	Event.no[5].Flag 										:= Diag_UnderVoltage OR Diag_OverVoltage OR Diag_NoControlPower;
	Event.no[6].Flag 										:= Diag_ShortCircuit OR Diag_ShortCircuitB OR Diag_OpenLoadA OR Diag_OpenLoadB; 
	Event.no[7].Flag 										:= Diag_Saturated;
	Event.no[8].Flag										:= Diag_OverTemperature ;
	Event.no[9].Flag 										:= ErrorLimitPos; 	
	Event.no[10].Flag 										:= ErrorLimitNeg;	
(*	Event.no[11].Flag 										:= FALSE; 				
	Event.no[12].Flag 										:= FALSE;					
	Event.no[13].Flag 										:= FALSE; 			Event.no[9].Class := TC2_SYSTEM.TCEVENTCLASS_WARNING;
	Event.no[14].Flag 										:= FALSE; 			Event.no[10].Class := TC2_SYSTEM.TCEVENTCLASS_WARNING;
	Event.no[15].Flag 										:= FALSE;
	Event.no[16].Flag 										:= FALSE;
	Event.no[17].Flag 										:= FALSE;
	Event.no[18].Flag 										:= FALSE;
	Event.no[19].Flag 										:= FALSE;
	Event.no[20].Flag 										:= FALSE;
	Event.no[21].Flag 										:= FALSE;
	Event.no[22].Flag 										:= FALSE;
	Event.no[23].Flag 										:= FALSE;
	Event.no[24].Flag 										:= FALSE;
	Event.no[25].Flag 										:= FALSE;
*)

(******************************************************************************)
END_METHOD

METHOD PUBLIC confirm : bool
VAR_INPUT
END_VAR
confirm			:= Event.confirm();
END_METHOD

END_FUNCTION_BLOCK

// POUs/IO/Drives/Stepper/AxDriveStepperParam
{attribute 'no_check'}
//FB template to read and write parameter
//The FB can be enherided and derivatived methods of SeqRead/SeqWrite used for application specific parameter.
//The extended methods need to call the super class at the beginning and return true if execution will be finished. The allowed states for new parameter are 1..99
//
//Calculating NC-parameter
//Sacling with Enc 		= Distance per revolution / (Increments x 4 fold)
//Scaling without Enc.  = Distance per revolution / (Fullsteps x Microsteps)
//Scalingfactor = 360° / (1024 x 4) OR 360° / (200 x 64) 
//
//Ref. Velocity = (Max. Outputfreq * Distance per rev.) / (Fullsteps * Microsteps)
//3515 °/s = (126kHz * 360°) / (200 * 64)
//Set kv to 0 to see whether ref. velocity is correct
//
FUNCTION_BLOCK AxDriveStepperParam EXTENDS AxRWParaBase
VAR_OUTPUT CONSTANT
END_VAR                                 					
VAR_INPUT                               					
	AdsAddr													: 	AMSADDR; //Terminal AMS Net Addr.                                        	                                        	
	Channel													:	USINT := 0; //Drive channel 0 or 1 
	SetKpPosition											:	LREAL; //0:8014:02 - only at EL70x7
	SetKpVelocity											:	LREAL; //0:8014:03 in 0.1mA/(rad/s) - at EL70x1 -> 0:8013:01 - at EL70x1
	SetKiVelocity											:	LREAL; //0:8013:02 in 0.001 - NOT for EL70x7
	SetTnVelocity											:	LREAL; //0:8014:04 in 0.01 ms - only at EL70x7 
	SetKpCurrent											:	LREAL; //0:8011:01 
	SetKiCurrent											:	LREAL; //0:8011:02 

	SetCalibrInvertDirForCamSearch							:	BOOL; 	//0:8021:13 / TRUE=Cam search direction negative
	SetCalibrInvertDirForOfCam								:	BOOL; 	//0:8021:14 / TRUE=Sync impuls (off cam) search direction negative
	SetCalibrPosition										:	UDINT;	//0:8020:08 
END_VAR 
VAR_IN_OUT
END_VAR                               					
VAR_OUTPUT
	DeviceType												:	STRING(15); //e.g. EL7037

	KpPosition												:	LREAL;
	KpVelocity												:	LREAL;
	KiVelocity												:	LREAL; //Not available at EL70x7
	TnVelocity												:	LREAL; //Only available at EL70x7
	KpCurrent												:	LREAL;
	KiCurrent												:	LREAL;	
	CalibrInvertDirForCamSearch								:	BOOL; // TRUE=Cam search direction negative
	CalibrInvertDirForOfCam									:	BOOL; // TRUE=Sync impuls (off cam) search direction negative
	CalibrPosition											:	UDINT;
END_VAR                         	
VAR
(* Cache ************************************************************)
	
(* Trigger **********************************************************)

(* Timer ******************************************************************)

(* FBs ***************************************************************)
	CoEWrite												: FB_EcCoESdoWriteEx := (tTimeout := DEFAULT_ADS_TIMEOUT);
	CoERead													: FB_EcCoeSdoReadEx := (tTimeout := DEFAULT_ADS_TIMEOUT);

(* Dummy memory **********************************************************)
END_VAR

	(* Read/Write stepper drive parameter												*)
	(************************************************************************************)

(* Execute ***************************************************************************************)
	SUPER^();
	
(*************************************************************************************************)

PROPERTY PROTECTED deviceAddrIsValid : BOOL
GET
deviceAddrIsValid := AdsAddr.port > 0;
END_GET
END_PROPERTY

METHOD PROTECTED getValue : BOOL //Return value = TRUE if execution finished and state incremented 
VAR_INPUT
	Index						:	WORD;
	SubIndex					:	BYTE;
	Len							:	UDINT;
	pActValue					:	PVOID; //Address of variable for actual value
	pSetValue					:	PVOID; //Address of variable for ser value variable, can be zero if no corresponding SetVariable exists
	CompleteAccess				:	BOOL;
END_VAR
CoERead(bExecute := TRUE , nIndex := Index ,nSubIndex := SubIndex ,pDstBuf := pActValue ,cbBufLen := Len, bCompleteAccess  := CompleteAccess);
IF NOT CoERead.bBUSY 	
THEN
	IF NOT CoERead.bError
	THEN
		IF pSetValue <> 0 THEN MEMCPY(pSetValue, pActValue, Len); END_IF
		state 												:= state + 1; 
	ELSE
		Busy												:= FALSE;
		Error												:= TRUE;
		ErrorId												:= CoERead.nErrId;
		ErrorText											:= CONCAT('Error read parameter in state:' , TO_STRING(state * -1));
		ErrorText											:= CONCAT(ErrorText , ' Id:');
		ErrorText											:= CONCAT(ErrorText , TO_STRING(ErrorId));
		State												:= 9999;
	END_IF
	CoERead(bExecute := FALSE);
	getValue												:= TRUE;
END_IF
END_METHOD

METHOD PROTECTED seqRead : BOOL //Return value = TRUE if execution finished 
VAR_IN_OUT
	State							:	INT;
END_VAR

(* Sequence read parameter **********************************)
	CASE state OF
	1..99: //Read application specific parameter  
		seqRead												:= TRUE;
		
	1001: (* Init step ******************************************************)
		CoERead(bExecute := FALSE, sNetId:= F_CreateAmsNetId(nIds := AdsAddr.netId), nSlaveAddr:= AdsAddr.port);
		IF NOT CoERead.bBusy
		THEN
			state											:= state + 1;	
		END_IF
		
	1002: (* Device name *************************************************************************************)
		IF LEN(DeviceType) > 0 AND NOT CoERead.bBusy
		THEN
			state											:= state + 1;
		ELSE
			getValue(Index:= 16#1008,	Subindex := 16#0,	LEN := SIZEOF(DeviceType),	pActValue := ADR(DeviceType),	pSetValue := 0, completeAccess := FALSE);
		END_IF

			
	1003: (* kp_current *************************************************************************************)
		IF DeviceType = 'EL7041-1000' OR DeviceType = 'EP7041-3002' OR DeviceType = 'EP7041-3102'
		THEN
			state											:= state + 1; (* NOT available *)
		ELSE	
			IF getValue(Index:= 16#8011,	Subindex := 16#01,	LEN := SIZEOF(_UINT),	pActValue := ADR(_UINT),	pSetValue := 0, completeAccess := FALSE)
			THEN
				KpCurrent := SetKpCurrent					:= SEL(Error, UINT_TO_LREAL(_UINT), 0.0);
			END_IF
		END_IF
		
	1004: (* ki current **********************************)
		IF DeviceType = 'EL7041-1000' OR DeviceType = 'EP7041-3002' OR DeviceType = 'EP7041-3102'
		THEN
			state											:= state + 1; (* Not available *)
		ELSE	
			IF getValue(Index:= 16#8011,	Subindex := 16#02,	LEN := SIZEOF(_UINT),	pActValue := ADR(_UINT),	pSetValue := 0, completeAccess := FALSE)
			THEN
				KiCurrent := SetKiCurrent					:= SEL(Error, UINT_TO_LREAL(_UINT), 0.0);
			END_IF		
		END_IF
	
	1005: (* Kp velocity ****************************************************************************************)
		IF DeviceType = 'EL7041-1000'
		THEN
			state											:= state + 1;
		ELSIF DeviceType = 'EL7037' OR DeviceType = 'EL7047' 
		THEN			
			IF getValue(Index:= 16#8014,	Subindex := 16#03,	LEN := SIZEOF(_UDINT),	pActValue := ADR(_UDINT),	pSetValue := 0, completeAccess := FALSE)
			THEN
				KpVelocity := SetKpVelocity					:= SEL(Error, UDINT_TO_LREAL(_UDINT), 0.0);
			END_IF
		ELSE			
			IF getValue(Index:= 16#8013,	Subindex := 16#01,	LEN := SIZEOF(_UINT),	pActValue := ADR(_UINT),	pSetValue := 0, completeAccess := FALSE)
			THEN
				KpVelocity := SetKpVelocity					:= SEL(Error, UINT_TO_LREAL(_UINT), 0.0);
			END_IF			
		END_IF	
		
	1006: (* Tn velocity or Ki Velocity ****************************************************************************************)
		IF DeviceType = 'EL7041-1000'
		THEN
			state											:= state + 1;
		ELSIF DeviceType = 'EL7037' OR DeviceType = 'EL7047'
		THEN (* Tn velocity*)			
			IF getValue(Index:= 16#8014,	Subindex := 16#04,	LEN := SIZEOF(_UINT),	pActValue := ADR(_UINT),	pSetValue := 0, completeAccess := FALSE)
			THEN
				KiVelocity := SetKiVelocity					:= SEL(Error, UINT_TO_LREAL(_UINT), 0.0);
			END_IF
			
		ELSE (* Ki Velccity*)
			IF getValue(Index:= 16#8013,	Subindex := 16#02,	LEN := SIZEOF(_UINT),	pActValue := ADR(_UINT),	pSetValue := 0, completeAccess := FALSE)
			THEN
				KiVelocity := SetKiVelocity					:= SEL(Error, UINT_TO_LREAL(_UINT), 0.0);
			END_IF
		END_IF 
	
	1007: (* Kp position ****************************************************************************************)
		IF DeviceType = 'EL7037' OR DeviceType = 'EL7047' 
		THEN			
			IF getValue(Index:= 16#8014,	Subindex := 16#02,	LEN := SIZEOF(_UINT),	pActValue := ADR(_UINT),	pSetValue := 0, completeAccess := FALSE)
			THEN
				KpPosition := SetKpPosition					:= SEL(Error, UINT_TO_LREAL(_UINT), 0.0);
			END_IF			
		ELSE
			;
		END_IF	
	
	1008: (* Homing cam search direction ****************************************************************************************)		
		IF DeviceType = 'EL7041-1000' 
		THEN
			state											:= state + 1;
		ELSE
			getValue(Index:= 16#8021,	Subindex := 16#13,	LEN := SIZEOF(CalibrInvertDirForCamSearch),	pActValue := ADR(CalibrInvertDirForCamSearch),	pSetValue := ADR(SetCalibrInvertDirForCamSearch), completeAccess := FALSE);			
		END_IF
	
	1009: (* Homing cam of direxction ****************************************************************************************)	
		IF DeviceType = 'EL7041-1000'
		THEN
			state											:= state + 1;
		ELSE
			getValue(Index:= 16#8021,	Subindex := 16#14,	LEN := SIZEOF(CalibrInvertDirForOfCam),	pActValue := ADR(CalibrInvertDirForOfCam),	pSetValue := ADR(SetCalibrInvertDirForOfCam), completeAccess := FALSE);			
		END_IF

	1010: (* Calibration value ****************************************************************************************)
		IF DeviceType = 'EL7041-1000'
		THEN
			state											:= state + 1;
		ELSE
			getValue(Index:= 16#8020,	Subindex := 16#08,	LEN := SIZEOF(CalibrPosition),	pActValue := ADR(CalibrPosition),	pSetValue := ADR(SetCalibrPosition), completeAccess := FALSE);			
		END_IF
		
	ELSE
		state												:= 1;
	END_CASE

(***********************************************************************************)
END_METHOD

METHOD PROTECTED seqWrite : BOOL //Return value = TRUE if execution finished 
VAR_IN_OUT
	State							:	INT;
END_VAR

(* Sequence write parameter *********************************************)
	CASE state OF
	1..99: //Write application specific parameter  
		seqWrite											:= TRUE;
		
	1001: (* Init step ******************************************************)
		CoEWrite(bExecute := FALSE, sNetId:= F_CreateAmsNetId(nIds := AdsAddr.netId), nSlaveAddr:= AdsAddr.port);
		IF NOT CoEWrite.bBusy
		THEN
			state											:= state + 1;	
		END_IF
		
	1002: (* Kv position *************************************************************************************)
		IF DeviceType = 'EL7041-1000' OR DeviceType = 'EP7041-3002' OR DeviceType = 'EP7041-3102'
			OR KpCurrent = SetKpCurrent AND NOT CoEWrite.bBusy
		THEN
			state											:= state + 1;
		ELSE
			_UINT											:= LREAL_TO_UINT(SetKpCurrent);
			IF setValue(Index:= 16#8011,	Subindex := 16#01,	LEN := SIZEOF(_UINT),		pActValue := 0,		pSetValue := ADR(_UINT) , completeAccess := FALSE)
			THEN
				KpCurrent									:= SetKpCurrent;
			END_IF			
		END_IF	
		
	1003: (* ki current **********************************)
		IF DeviceType = 'EL7041-1000' OR DeviceType = 'EP7041-3002' OR DeviceType = 'EP7041-3102'
			OR KiCurrent = SetKiCurrent AND NOT CoEWrite.bBusy
		THEN
			state											:= state + 1;
		ELSE
			_UINT											:= LREAL_TO_UINT(SetKiCurrent);
			IF setValue(Index:= 16#8011,	Subindex := 16#02,	LEN := SIZEOF(_UINT),		pActValue := 0,		pSetValue := ADR(_UINT) , completeAccess := FALSE)
			THEN
				KiCurrent									:= SetKiCurrent;
			END_IF			
		END_IF
	
	1004: (* Kp velocity ****************************************************************************************)
		IF DeviceType = 'EL7041-1000' 
			OR KpVelocity = SetKpVelocity AND NOT CoEWrite.bBusy
		THEN
			state											:= state + 1;
		ELSE
			IF DeviceType = 'EL7037' OR DeviceType = 'EL7047' 
			THEN
				_UDINT										:=LREAL_TO_UDINT(SetKpVelocity);
				IF setValue(Index:= 16#8014,	Subindex := 16#03,	LEN := SIZEOF(_UDINT),		pActValue := 0,		pSetValue := ADR(_UDINT) , completeAccess := FALSE)
				THEN
					KpVelocity								:= SetKpVelocity;
				END_IF	
			ELSE
				_UINT										:=LREAL_TO_UINT(SetKpVelocity);
				IF setValue(Index:= 16#8013,	Subindex := 16#01,	LEN := SIZEOF(_UINT),		pActValue := 0,		pSetValue := ADR(_UINT) , completeAccess := FALSE)
				THEN
					KpVelocity								:= SetKpVelocity;
				END_IF	
			END_IF		
		END_IF
	
	1005: (* Tn velocity or Ki velocity****************************************************************************************)
		IF SetTnVelocity = TnVelocity AND SetKiVelocity = KiVelocity AND NOT CoEWrite.bBusy OR DeviceType = 'EL7041-1000'
		THEN 
			state											:= state + 1;
		ELSE
			IF DeviceType = 'EL7037' OR DeviceType = 'EL7047' 
			THEN (* Tn Velocity *)
				_UINT										:= LREAL_TO_UINT(SetTnVelocity);
				IF setValue(Index:= 16#8014,	Subindex := 16#04,	LEN := SIZEOF(_UINT),		pActValue := 0,		pSetValue := ADR(_UINT) , completeAccess := FALSE)
				THEN
					TnVelocity								:= SetTnVelocity;
				END_IF	
				
	
			ELSE (* Ki Velocity *)
				_UINT										:= LREAL_TO_UINT(SetKiVelocity);
				IF setValue(Index:= 16#8013,	Subindex := 16#02,	LEN := SIZEOF(_UINT),		pActValue := 0,		pSetValue := ADR(_UINT) , completeAccess := FALSE)
				THEN
					KiVelocity								:= SetKiVelocity;
				END_IF				
			END_IF	
		END_IF
	
	1006: (* Kp position ****************************************************************************************)		
		IF SetKpPosition <> KpPosition AND (DeviceType = 'EL7037' OR DeviceType = 'EL7047')
		THEN
			_UINT											:= LREAL_TO_UINT(SetKpPosition);
			IF setValue(Index:= 16#8014,	Subindex := 16#02,	LEN := SIZEOF(_UINT),		pActValue := 0 ,		pSetValue := ADR(_UINT) , completeAccess := FALSE)	
			THEN
				KpPosition									:= SetKpPosition;
			END_IF			
		ELSIF NOT CoEWrite.bBusy
		THEN
			state											:= state + 1;
		END_IF
			
	1007: (* Homing cam search direction ********************************************************************************************)
		IF DeviceType = 'EL7041-1000' 
		THEN
			state											:= state + 1;
		ELSE
			setValue(Index:= 16#8021,	Subindex := 16#13,	LEN := SIZEOF(SetCalibrInvertDirForCamSearch),		pActValue := ADR(CalibrInvertDirForCamSearch) ,		pSetValue := ADR(SetCalibrInvertDirForCamSearch) , completeAccess := FALSE);
		END_IF
		
	1008: (* Homing cam of direction *****************************************************************************************)
		IF DeviceType = 'EL7041-1000' 
		THEN
			state											:= state + 1;
		ELSE
			setValue(Index:= 16#8021,	Subindex := 16#14,	LEN := SIZEOF(SetCalibrInvertDirForOfCam),		pActValue := ADR(CalibrInvertDirForOfCam) ,		pSetValue := ADR(SetCalibrInvertDirForOfCam) , completeAccess := FALSE)	;	
		END_IF
	
	1009: (* Calibration position ***********************************************************************)	
		IF DeviceType = 'EL7041-1000' 
		THEN
			state											:= state + 1;
		ELSE
			setValue(Index:= 16#8020,	Subindex := 16#08,	LEN := SIZEOF(SetCalibrPosition),		pActValue := ADR(CalibrPosition) ,		pSetValue := ADR(SetCalibrPosition) , completeAccess := FALSE)	;	
		END_IF
	ELSE
		state												:= 1;
	END_CASE

(************************************************************************************)
END_METHOD

METHOD PROTECTED setValue : BOOL //Return value = TRUE if execution finished and state incremented 
VAR_INPUT
	Index						:	Word;
	SubIndex					:	BYTE;
	Len							:	UDINT;
	pActValue					:	PVOID; //Address of variable for actual value, can be zero if no corresponding acual value variable exists
	pSetValue					:	PVOID; //Address of variable for set value variable
	CompleteAccess				:	BOOL;
END_VAR


IF pActValue <> 0 AND pSetValue <> 0 AND_THEN MEMCMP(pSetValue, pActValue, Len) = 0
THEN //Skip write parameter if set and actual value are equel
	state													:= state + 1;	
	setValue												:= TRUE;
ELSE
	CoEWrite(bExecute := TRUE, nIndex := Index ,nSubIndex := SubIndex , pSrcBuf := pSetValue ,cbBufLen := Len , bCompleteAccess := CompleteAccess );
	IF NOT CoEWrite.bBusy
	THEN
		IF NOT CoEWrite.bError
		THEN
			IF pActValue <> 0 THEN MEMCPY(pActValue, pSetValue, Len); END_IF	
			state											:= state + 1;
		ELSE
			Busy											:= FALSE;
			Error											:= TRUE;
			ErrorId											:= CoEWrite.nErrId;
			ErrorText										:= CONCAT('Error write parameter in state:' , TO_STRING(state * -1));
			ErrorText										:= CONCAT(ErrorText , ' Id:');
			ErrorText										:= CONCAT(ErrorText , TO_STRING(ErrorId));
			State											:= 9999;
		END_IF
		CoEWrite(bExecute := FALSE);
		setValue											:= TRUE;
	END_IF		
END_IF
END_METHOD

END_FUNCTION_BLOCK

// POUs/IO/Drives/AxDriveGetRef
{attribute 'no_check'}
//Provides drive reference (Ref -> ST_DriveRef) based on NC-AxisID
//Drive reference is needed for FB's of lib Drive e.g. FB_SoEAX5000FirmwareUpdate_ByDriveRef
FUNCTION_BLOCK AxDriveGetRef EXTENDS FbBase
VAR CONSTANT                								
	NCIDXG_AXPARMS											: UDINT := 16#0000_4000;	(* Axis with ID: Parameter 			*)
	NCIDXO_AXP_HWAMSADDR									: UDINT := 16#0000_0031;	
	MIN_ADSREAD_BUFFER										:	INT := 0;
	MAX_ADSREAD_BUFFER										:	INT := 9;
END_VAR 
VAR_INPUT                   					
	AmsNetId												: T_AmsNetId := '';	(* netID of PC with NC *)			      
	AxisId													:	DWORD; //NC axis id	
END_VAR
VAR_OUTPUT                  								
	DriveAmsNetId											: T_AmsNetIdArr; (* Ams net id as array of bytes *)
    DriveRef												: ST_DriveRef; 	(* contains sNetID of EcMaster, nSlaveAddr of EcDrive, nDriveNo of EcDrive, either preset or read from NC *)
END_VAR              								                 								
VAR                         								
(* cache ********************************************)
	AdsReadBuffer											: ARRAY[MIN_ADSREAD_BUFFER..MAX_ADSREAD_BUFFER] OF BYTE;
                						
(* trigger ******************************************)

(* timer ********************************************)
	
(* blocks *******************************************)	
	AdsRead													: ADSREAD := (TMOUT := DEFAULT_ADS_TIMEOUT);
	
(* dummys *******************************************)
END_VAR

	(* Create drive ref for device 									*)
	(****************************************************************)

(* Sequence ****************************************)
	rtExecute(CLK := Execute);
	CASE state OF 
	0:	
		Busy												:= FALSE;
		IF NOT Execute
		THEN
			Done											:= FALSE;
			Error											:= FALSE;
			ErrorId											:= 0;
		ELSIF rtExecute.Q
		THEN
			Busy											:= TRUE;
			Done											:= FALSE;
			Error											:= FALSE;
			ErrorId											:= 0;
			AdsRead(READ := FALSE);
			MEMSET(ADR(DriveRef), 0, SIZEOF(DriveRef));
			MEMSET(ADR(AdsReadBuffer), 0, SIZEOF(AdsReadBuffer));
			state											:= State + 1;
		END_IF 
	
	1: //Get drive slave address
		AdsRead(
			NETID	:= AmsNetId,
			PORT	:= AMSPORT_R0_NC,
			IDXGRP	:= NCIDXG_AXPARMS + AxisId,
			IDXOFFS	:= NCIDXO_AXP_HWAMSADDR,
			LEN		:= SIZEOF(AdsReadBuffer) ,
			DESTADDR:= ADR(AdsReadBuffer),
			READ	:= TRUE);
		IF NOT AdsRead.BUSY
		THEN
			IF NOT AdsRead.ERR 
			THEN
				MEMCPY(ADR(DriveAmsNetId), ADR(AdsReadBuffer), SIZEOF(DriveAmsNetId)); 							(* AdsreadBuffer[0..5] *)
				MEMCPY(ADR(DriveRef.nSlaveAddr), ADR(AdsReadBuffer[6]), SIZEOF(DriveRef.nSlaveAddr));  	(* AdsreadBuffer[6..7] *)
				MEMCPY(ADR(DriveRef.nDriveNo), ADR(AdsReadBuffer[8]), SIZEOF(DriveRef.nDriveNo));  		(* AdsreadBuffer[8..9] *)

				(* create string out of byte array *)
				DriveRef.sNetId 							:= F_CreateAmsNetId(DriveAmsNetId);
				
				Busy										:= FALSE;
				Done										:= TRUE;
				state										:= 0;
			ELSE
				Busy										:= FALSE;
				Error										:= TRUE;
				ErrorId										:= AdsRead.ERRID;
				State										:= 0;
			END_IF
		END_IF
	END_CASE
	
(**********************************************************************************)

END_FUNCTION_BLOCK

// POUs/IO/EL-EP/EL3403/EL3403
{attribute 'no_check'}
FUNCTION_BLOCK EL3403 Extends EcSlaveInfoData
VAR CONSTANT
	MIN_PHASE												:	INT := 1;
	MAX_PHASE												:	INT := 3;
END_VAR  
VAR_INPUT
	IndexOut										AT %Q*	:	ARRAY[MIN_PHASE..MAX_PHASE] OF USINT;
	Transmission											:	ARRAY[MIN_PHASE..MAX_PHASE] OF LREAL;	//Transmission current transformator for each phase e.g. 750 *)
END_VAR
VAR_OUTPUT
	(* Inputs Channel 1-3 *)
	TxPDOToggle										AT %I*	: 	ARRAY[MIN_PHASE..MAX_PHASE] OF BOOL;
	IndexIn											AT %I*	: 	ARRAY[MIN_PHASE..MAX_PHASE] OF USINT;
	Current													: 	ARRAY[MIN_PHASE..MAX_PHASE] OF LREAL; 	//Unit: 0,000001 A
	Voltage													: 	ARRAY[MIN_PHASE..MAX_PHASE] OF LREAL; 	//Unit: 0,0001 V
	ActivePower												: 	ARRAY[MIN_PHASE..MAX_PHASE] OF LREAL; 	//Unit: 0,01 W

	(* PM Status Data *)
	MissingZeroCrossingA							AT %I*	: 	BOOL;
	MissingZeroCrossingB							AT %I* 	: 	BOOL;
	MissingZeroCrossingC							AT %I* 	: 	BOOL;
	PhaseSequenceError								AT %I* 	: 	BOOL;
//	SyncError										AT %I* 	: 	BOOL;
                                                              	
	(* MultiplexValues	*)
	ApparentPower											:	ARRAY[MIN_PHASE..MAX_PHASE] OF LREAL; 	//apparent power unit: 0,01 VA
	ReactivePower											:	ARRAY[MIN_PHASE..MAX_PHASE] OF LREAL; 	//reactive power unit: 0,01 VAr
	PowerFactor												:	ARRAY[MIN_PHASE..MAX_PHASE] OF LREAL; 	//effective power cos phi Unit: 0,001
	EnergyConsumption										:	ARRAY[MIN_PHASE..MAX_PHASE] OF LREAL; 	//energy unit: 0,001 Wh
	EnergyConsumptionInvers									:	ARRAY[MIN_PHASE..MAX_PHASE] OF LREAL; 	//energy unit: 0,001 Wh
	TimestampDistClocks										:	ARRAY[MIN_PHASE..MAX_PHASE] OF LREAL; 	//timestamp unit : 1 ns
	Frequency												:	ARRAY[MIN_PHASE..MAX_PHASE] OF LREAL; 	//frequenzy unit : 0,1 Hz

END_VAR
VAR (* Internal IOs *)
	_Current										AT %I* 	: 	ARRAY[MIN_PHASE..MAX_PHASE] OF DINT; 	//Unit: 0,000001 A
	_Voltage										AT %I* 	: 	ARRAY[MIN_PHASE..MAX_PHASE] OF DINT; 	//Unit: 0,0001 V
	_ActivePower									AT %I* 	: 	ARRAY[MIN_PHASE..MAX_PHASE] OF DINT; 	//Unit: 0,01 W

	_VariantValue									AT %I* 	: 	ARRAY[MIN_PHASE..MAX_PHASE] OF DINT;
//	_SyncErrorChannel								AT %I* 	: 	ARRAY[MIN_PHASE..MAX_PHASE] OF BOOL; 	//reserved
//	_SyncErrorTerminal										: 	BOOL;	//reserved
END_VAR                       							
VAR
	i														:	INT;
END_VAR

(* EL 3403 IO 									*)
(************************************************)

(* Get Index Values *****************************)
	FOR i := MIN_PHASE TO MAX_PHASE DO
		Current[i]											:= Transmission[i] * DINT_TO_LREAL(_Current[i]) / 1000000.0; //A
		Voltage[i]											:= (*Uebersetzung[i] **) DINT_TO_LREAL(_Voltage[i]) / 10000.0; //V
		ActivePower[i]										:= Transmission[i] * DINT_TO_LREAL(_ActivePower[i]) / 100.0; //W
                                            				
		CASE IndexIn[i] OF                  				
		0:(*Scheinleistung*)                				
			ApparentPower[i]								:= Transmission[i] * DINT_TO_LREAL(_VariantValue[i]) / 100.0; //VA
                                            				
		1:(*Blindleistung*)                 				
			ReactivePower[i]								:= Transmission[i] * DINT_TO_LREAL(_VariantValue[i]) / 100.0; //VAr
                                            				
		2:(*Energie*)                       				
			EnergyConsumption[i]							:= Transmission[i] * DINT_TO_LREAL(_VariantValue[i]) / 1000.0; //Wh
                                            				
		3:(*Wirkleistungsfaktor*)           				
			PowerFactor[i]									:= DINT_TO_LREAL(_VariantValue[i]) / 1000.0; //cos phi
                                            				
		4:(*Frequenz*)                      	
			Frequency[i]									:= DINT_TO_LREAL(_VariantValue[i]) / 10.0; //Hz
                                            				
		5:(*Energie Invers*)                				
			EnergyConsumptionInvers[i]						:= Transmission[i] * DINT_TO_LREAL(_VariantValue[i]) / 1000.0;
                                            				
		100:(*Zeitstempel*)                 				
			TimestampDistClocks[i]							:= DINT_TO_LREAL(_VariantValue[i]);
	
		END_CASE

	END_FOR

(***********************************************)

END_FUNCTION_BLOCK

// POUs/IO/EL-EP/EL3403/EL3403Logic
{attribute 'no_check'}
//FB gets raw data from EL3404 every cycle and calculate real values *)
FUNCTION_BLOCK EL3403Logic
VAR_INPUT
	TrigReadVariantValues									:	BOOL 	:= FALSE;	//Rising edge reports actual total values on FB outputs
	Transmission											:	LREAL 	:= 750.0; 	//Transmission current transformator
	Mode													:	INT 	:= 0; 		(* 	0 = Phase 1-3
																					  	1 = Phase 1
																					 	2 = Phase 2
																					 	3 = Phase 3 *)                                   						
END_VAR                             	
VAR_OUTPUT
	(* Components OUTPUT -> ReadOnly ! *)
	IO														:	EL3403;
                                    				                                					
	(* Total Values *)              					
	TotalEffectivePower										: 	LREAL; 	//W
	TotalPowerFactor										: 	LREAL; 	//total power factor cos phi
	TotalEnergyConsumption									: 	LREAL; 	//Wh
                                    					
	(* Error *)                     					
	ErrorPhaseSequence										:	BOOL;
	ErrorMissingZeroCrossing								:	BOOL;
	TimeStart												: 	TIME;		(* Startzeit *)
	TimeEnd													: 	TIME;		(* Endzeit *)
	TimeDiff												: 	TIME;		(* Differenz Start End *)
	
	(* Ctrl Status  *)              					
	Valid													:	BOOL;	//TRUE when data is valid
	Busy													:	BOOL;	//Busy is TRUE at the rising edge of Execute and FALSE when one of the outputs Done, Aborted, or Error is set 
	Error													:	BOOL;	//Rising edge of Error informs that an error occurred during the execution of the Function Block 

END_VAR                             	
VAR                                 	
	rtReadVariantValues										:	R_Trig;
	state													:	INT;
	_MIN_PHASE												:	INT;
	_MAX_PHASE												:	INT;
	i														:	INT;
END_VAR

(* Work EL3403 data 						*)
(********************************************)

(* Work Termianl IO ******************************************)
	FOR i := IO.MIN_PHASE TO IO.MAX_PHASE 
	DO
		IO.Transmission[i] 									:= Transmission;
	END_FOR

	IO();

(* Error *****************************************************)
	Error 													:= IO.WCState OR IO.InfoDataState <> Tc2_EtherCAT.EC_DEVICE_STATE_OP;

(* Get Total Values ******************************************)
IF NOT Error
THEN
	CASE Mode OF
	1:
		TotalEffectivePower 								:= IO.ActivePower[1];
		TotalPowerFactor 									:= IO.PowerFactor[1];
		TotalEnergyConsumption 								:= IO.EnergyConsumption[1];
	2:                              						
		TotalEffectivePower 								:= IO.ActivePower[2];
		TotalPowerFactor 									:= IO.PowerFactor[2];
		TotalEnergyConsumption 								:= IO.EnergyConsumption[2];
	3:                              						
		TotalEffectivePower 								:= IO.ActivePower[3];
		TotalPowerFactor 									:= IO.PowerFactor[3];
		TotalEnergyConsumption 								:= IO.EnergyConsumption[3];
	ELSE (* Phase 1-3 *)            						
		TotalEffectivePower 								:= IO.ActivePower[1] + IO.ActivePower[2] + IO.ActivePower[3];
		TotalPowerFactor 									:= (IO.PowerFactor[1] + IO.PowerFactor[2] + IO.PowerFactor[3]) / 3.0;
		TotalEnergyConsumption 								:= IO.EnergyConsumption[1] + IO.EnergyConsumption[2] + IO.EnergyConsumption[3];
	END_CASE                        	

END_IF

(* Trigger ReadVariantValues ******************************)
rtReadVariantValues(CLK := TrigReadVariantValues);

IF rtReadVariantValues.Q
	OR state <> 0
THEN
	ReadVariantValues(Mode := Mode);
END_IF

(********************************************************)

METHOD PUBLIC readVariantValues : Bool //Return value = TRUE if busy
VAR_INPUT
	Mode								:	INT 	:= 0; (* 	0 = Phase 1-3
															  		1 = Phase 1
															 	 	2 = Phase 2
															 		3 = Phase 3 *)
END_VAR
IF state = 0 
THEN
	THIS^.Mode												:= Mode;
	CASE mode OF
	1:
		_MIN_PHASE 											:= IO.MIN_PHASE;
		_MAX_PHASE 											:= IO.MIN_PHASE;
	2:             											
		_MIN_PHASE 											:= IO.MIN_PHASE + 1;
		_MAX_PHASE 											:= IO.MIN_PHASE + 1;
	3:             											
		_MIN_PHASE 											:= IO.MAX_PHASE;
		_MAX_PHASE 											:= IO.MAX_PHASE;
	ELSE           											
		_MIN_PHASE 											:= IO.MIN_PHASE;
		_MAX_PHASE 											:= IO.MAX_PHASE;
	END_CASE
	state 													:= 1;
	TimeStart 												:= TIME();
END_IF

(* Read Variant Values *******************************)
	CASE state OF
	0:
		;
		
	1:
		FOR i := _MIN_PHASE TO _MAX_PHASE DO
			IO.IndexOut[i] 									:= 0;
			IF IO.IndexIn[i] = IO.IndexOut[i]
				AND i = _MAX_PHASE
			THEN (* Set Next index *)
				state 										:= 2;
			ELSE
				;
			END_IF
		END_FOR

	2:
		FOR i := _MIN_PHASE TO _MAX_PHASE DO
			IO.IndexOut[i] 									:= 1;
			IF IO.IndexIn[i] = IO.IndexOut[i]
				AND i = _MAX_PHASE
			THEN (* Set Next index *)
				state 										:= 3;
			ELSE
				;
			END_IF
		END_FOR
	3:
		FOR i := _MIN_PHASE TO _MAX_PHASE DO
			IO.IndexOut[i] 									:= 2;
			IF IO.IndexIn[i] = IO.IndexOut[i]
				AND i = _MAX_PHASE
			THEN (* Set Next index *)
				state 										:= 4;
			ELSE
				;
			END_IF
		END_FOR
	4:
		FOR i := _MIN_PHASE TO _MAX_PHASE DO
			IO.IndexOut[i] 									:= 3;
			IF IO.IndexIn[i] = IO.IndexOut[i]
				AND i = _MAX_PHASE
			THEN (* Set Next index *)
				state 										:= 5;
			ELSE
				;
			END_IF
		END_FOR
	5:
		FOR i := _MIN_PHASE TO _MAX_PHASE DO
			IO.IndexOut[i] 									:= 4;
			IF IO.IndexIn[i] = IO.IndexOut[i]
				AND i = _MAX_PHASE
			THEN (* Set Next index *)
				state 										:= 6;
			ELSE
				;
			END_IF
		END_FOR

	6:
		FOR i := _MIN_PHASE TO _MAX_PHASE DO
			IO.IndexOut[i] 									:= 5;
			IF IO.IndexIn[i] = IO.IndexOut[i]
				AND i = _MAX_PHASE
			THEN (* Set Next index *)
				state 										:= 7;
			ELSE
				;
			END_IF
		END_FOR

	7:
		FOR i := _MIN_PHASE TO _MAX_PHASE DO
			IO.IndexOut[i] 									:= 100;
			IF IO.IndexIn[i] = IO.IndexOut[i]
				AND i = _MAX_PHASE
			THEN (* Set Next index *)
				Valid 										:= TRUE;
				state 										:= 0;
				TimeEnd 									:= TIME();
				TimeDiff 									:= TimeEnd - TimeStart;
			ELSE
				;
			END_IF
		END_FOR

	END_CASE
	
	Busy													:= state <> 0;
	ReadVariantValues 										:= Busy;
END_METHOD

END_FUNCTION_BLOCK

// POUs/IO/EL-EP/EL9x/EL9501
{attribute 'no_check'}
FUNCTION_BLOCK EL9501 EXTENDS EcSlaveInfoDataExt
VAR_INPUT
	SetVoltage					AT %Q*		:	REAL; // 0.0 - 20.0 [V]
END_VAR                 					 	
VAR_OUTPUT    
	{attribute 'displaymode':='binary'}             	
	Status						AT  %I*		:	WORD; // Terminal status (2 bytes)
          					 	
	Voltage								 	: 	AnalogInREAL ; 
	Current								 	: 	AnalogInREAL;
END_VAR                                 
VAR                                     

END_VAR

	(* EL9501 Power supply terminal	 0-20V	*)
	(****************************************)
	SUPER^();
	
(* Work objects *****************************)
	Voltage();
	Current();

(********************************************)

{attribute 'monitoring' := 'call'}
PROPERTY PUBLIC error : BOOL
GET
Error				:= Status.6 OR Voltage.Error OR Current.Error;
END_GET
END_PROPERTY

METHOD PUBLIC off : BOOL
VAR_INPUT
END_VAR
Off := CAM(SetVoltage, Voltage.Q, 0.01);
END_METHOD

{attribute 'monitoring' := 'call'}
PROPERTY PUBLIC overload : BOOL
GET
Overload 			:= Status.1;
END_GET
END_PROPERTY

{attribute 'monitoring' := 'call'}
PROPERTY PUBLIC overrange : BOOL
GET
Overrange 			:= Status.3;
END_GET
END_PROPERTY

{attribute 'monitoring' := 'call'}
PROPERTY PUBLIC underrange : BOOL
GET
Underrange 			:= Status.2;
END_GET
END_PROPERTY

{attribute 'monitoring' := 'call'}
PROPERTY PUBLIC warning : BOOL
GET
Warning 			:= Status.5;
END_GET
END_PROPERTY

END_FUNCTION_BLOCK

// POUs/IO/EL-EP/EL9x/EL9576
{attribute 'no_check'}
//EL Brake Chopper IOs
FUNCTION_BLOCK EL9576 
VAR_OUTPUT CONSTANT
END_VAR
VAR_INPUT
END_VAR
VAR_OUTPUT	
	Overtemperature									AT  %I* : BOOL;		//TRUE when there is an overtemperature on the PCB
	I2T_Error										AT  %I* : BOOL;		//TRUE when there is an overtemperature in the external resistor
	I2T_Warning										AT  %I* : BOOL;		//TRUE when the warning temperature threshold value from the CoE data has been exceeded
	Overvoltage										AT  %I* : BOOL;		//TRUE when the overvoltage threshold value has been exceeded
	Undervoltage									AT  %I* : BOOL;		//TRUE when the voltage has fallen below the undervoltage threshold value from the CoE data
	CopperOn										AT  %I* : BOOL;		//TRUE when the external resistor is active, i.e. electrical energy is being converted to thermal energy in the resistor
	OvercurrentProtection							AT  %I* : BOOL;		//TRUE when the external resistor is active, i.e. electrical energy is being converted to thermal energy in the resistor
	InputCycleCounter								AT  %I* : USINT;	//TRUE if the overcurrent or short-circuit detection of the EL9576 has been triggered. Otherwise the bit is permanently FALSE.
	DCLinkVoltage									AT  %I* : UDINT;	//External supply voltage in mV
	ResistorCurrent									AT  %I* : DINT;		//Current through the external resistor in mA
	DutyCycle										AT  %I* : USINT;	//Temporal utilization of the external resistor in the last 100 ms in %
	I2TLoadFactor									AT  %I* : USINT;	

	WcState											AT  %I* : BOOL;
	InputToggle										AT  %I* : BOOL;
	{attribute 'displaymode':='hex'}  
	State											AT  %I* : UINT;
	
END_VAR
VAR
{attribute 'hide'}
END_VAR

(* Ax_BrakeCopperIO						*)
(****************************************)
	
(* Work objects ****************************************)
	;
(*******************************************************)

END_FUNCTION_BLOCK

// POUs/IO/EL-EP/EL9x/EL95xxPowerTerminal
{attribute 'no_check'}
FUNCTION_BLOCK EL95xxPowerTerminal 
VAR_OUTPUT CONSTANT
END_VAR
VAR_INPUT
END_VAR
VAR_OUTPUT	
	PowerOK			 									AT  %I* : BOOL;
	Overload											AT  %I* : BOOL;
END_VAR
VAR
END_VAR

